    TEXT488 : BOOL ;	//TEXT N.488
    TEXT505 : BOOL ;	//TEXT N.505
    TEXT506 : BOOL ;	//TEXT N.506
    TEXT507 : BOOL ;	//TEXT N.507
    TEXT508 : BOOL ;	//TEXT N.508
    TEXT509 : BOOL ;	//TEXT N.509
    TEXT510 : BOOL ;	//TEXT N.510
    TEXT511 : BOOL ;	//TEXT N.511
    TEXT512 : BOOL ;	//TEXT N.512
    TEXT497 : BOOL ;	//TEXT N.497
    TEXT498 : BOOL ;	//TEXT N.498
    TEXT499 : BOOL ;	//TEXT N.499
    TEXT500 : BOOL ;	//TEXT N.500
    TEXT501 : BOOL ;	//TEXT N.501
    TEXT502 : BOOL ;	//TEXT N.502
    TEXT503 : BOOL ;	//TEXT N.503
    TEXT504 : BOOL ;	//TEXT N.504
    TEXT521 : BOOL ;	//TEXT N.521
    TEXT522 : BOOL ;	//TEXT N.522
    TEXT523 : BOOL ;	//TEXT N.523
    TEXT524 : BOOL ;	//TEXT N.524
    TEXT525 : BOOL ;	//TEXT N.525
    TEXT526 : BOOL ;	//TEXT N.526
    TEXT527 : BOOL ;	//TEXT N.527
    TEXT528 : BOOL ;	//TEXT N.528
    TEXT513 : BOOL ;	//TEXT N.513
    TEXT514 : BOOL ;	//TEXT N.514
    TEXT515 : BOOL ;	//TEXT N.515
    TEXT516 : BOOL ;	//TEXT N.516
    TEXT517 : BOOL ;	//TEXT N.517
    TEXT518 : BOOL ;	//TEXT N.518
    TEXT519 : BOOL ;	//TEXT N.519
    TEXT520 : BOOL ;	//TEXT N.520
    TEXT537 : BOOL ;	//TEXT N.537
    TEXT538 : BOOL ;	//TEXT N.538
    TEXT539 : BOOL ;	//TEXT N.539
    TEXT540 : BOOL ;	//TEXT N.540
    TEXT541 : BOOL ;	//TEXT N.541
    TEXT542 : BOOL ;	//TEXT N.542
    TEXT543 : BOOL ;	//TEXT N.543
    TEXT544 : BOOL ;	//TEXT N.544
    TEXT529 : BOOL ;	//TEXT N.529
    TEXT530 : BOOL ;	//TEXT N.530
    TEXT531 : BOOL ;	//TEXT N.531
    TEXT532 : BOOL ;	//TEXT N.532
    TEXT533 : BOOL ;	//TEXT N.533
    TEXT534 : BOOL ;	//TEXT N.534
    TEXT535 : BOOL ;	//TEXT N.535
    TEXT536 : BOOL ;	//TEXT N.536
    TEXT553 : BOOL ;	//TEXT N.553
    TEXT554 : BOOL ;	//TEXT N.554
    TEXT555 : BOOL ;	//TEXT N.555
    TEXT556 : BOOL ;	//TEXT N.556
    TEXT557 : BOOL ;	//TEXT N.557
    TEXT558 : BOOL ;	//TEXT N.558
    TEXT559 : BOOL ;	//TEXT N.559
    TEXT560 : BOOL ;	//TEXT N.560
    TEXT545 : BOOL ;	//TEXT N.545
    TEXT546 : BOOL ;	//TEXT N.546
    TEXT547 : BOOL ;	//TEXT N.547
    TEXT548 : BOOL ;	//TEXT N.548
    TEXT549 : BOOL ;	//TEXT N.549
    TEXT550 : BOOL ;	//TEXT N.550
    TEXT551 : BOOL ;	//TEXT N.551
    TEXT552 : BOOL ;	//TEXT N.552
    TEXT569 : BOOL ;	//TEXT N.569
    TEXT570 : BOOL ;	//TEXT N.570
    TEXT571 : BOOL ;	//TEXT N.571
    TEXT572 : BOOL ;	//TEXT N.572
    TEXT573 : BOOL ;	//TEXT N.573
    TEXT574 : BOOL ;	//TEXT N.574
    TEXT575 : BOOL ;	//TEXT N.575
    TEXT576 : BOOL ;	//TEXT N.576
    TEXT561 : BOOL ;	//TEXT N.561
    TEXT562 : BOOL ;	//TEXT N.562
    TEXT563 : BOOL ;	//TEXT N.563
    TEXT564 : BOOL ;	//TEXT N.564
    TEXT565 : BOOL ;	//TEXT N.565
    TEXT566 : BOOL ;	//TEXT N.566
    TEXT567 : BOOL ;	//TEXT N.567
    TEXT568 : BOOL ;	//TEXT N.568
    TEXT585 : BOOL ;	//TEXT N.585
    TEXT586 : BOOL ;	//TEXT N.586
    TEXT587 : BOOL ;	//TEXT N.587
    TEXT588 : BOOL ;	//TEXT N.588
    TEXT589 : BOOL ;	//TEXT N.589
    TEXT590 : BOOL ;	//TEXT N.590
    TEXT591 : BOOL ;	//TEXT N.591
    TEXT592 : BOOL ;	//TEXT N.592
    TEXT577 : BOOL ;	//TEXT N.577
    TEXT578 : BOOL ;	//TEXT N.578
    TEXT579 : BOOL ;	//TEXT N.579
    TEXT580 : BOOL ;	//TEXT N.580
    TEXT581 : BOOL ;	//TEXT N.581
    TEXT582 : BOOL ;	//TEXT N.582
    TEXT583 : BOOL ;	//TEXT N.583
    TEXT584 : BOOL ;	//TEXT N.584
    TEXT601 : BOOL ;	//TEXT N.601
    TEXT602 : BOOL ;	//TEXT N.602
    TEXT603 : BOOL ;	//TEXT N.603
    TEXT604 : BOOL ;	//TEXT N.604
    TEXT605 : BOOL ;	//TEXT N.605
    TEXT606 : BOOL ;	//TEXT N.606
    TEXT607 : BOOL ;	//TEXT N.607
    TEXT608 : BOOL ;	//TEXT N.608
    TEXT593 : BOOL ;	//TEXT N.593
    TEXT594 : BOOL ;	//TEXT N.594
    TEXT595 : BOOL ;	//TEXT N.595
    TEXT596 : BOOL ;	//TEXT N.596
    TEXT597 : BOOL ;	//TEXT N.597
    TEXT598 : BOOL ;	//TEXT N.598
    TEXT599 : BOOL ;	//TEXT N.599
    TEXT600 : BOOL ;	//TEXT N.600
    TEXT617 : BOOL ;	//TEXT N.617
    TEXT618 : BOOL ;	//TEXT N.618
    TEXT619 : BOOL ;	//TEXT N.619
    TEXT620 : BOOL ;	//TEXT N.620
    TEXT621 : BOOL ;	//TEXT N.621
    TEXT622 : BOOL ;	//TEXT N.622
    TEXT623 : BOOL ;	//TEXT N.623
    TEXT624 : BOOL ;	//TEXT N.624
    TEXT609 : BOOL ;	//TEXT N.609
    TEXT610 : BOOL ;	//TEXT N.610
    TEXT611 : BOOL ;	//TEXT N.611
    TEXT612 : BOOL ;	//TEXT N.612
    TEXT613 : BOOL ;	//TEXT N.613
    TEXT614 : BOOL ;	//TEXT N.614
    TEXT615 : BOOL ;	//TEXT N.615
    TEXT616 : BOOL ;	//TEXT N.616
    TEXT633 : BOOL ;	//TEXT N.633
    TEXT634 : BOOL ;	//TEXT N.634
    TEXT635 : BOOL ;	//TEXT N.635
    TEXT636 : BOOL ;	//TEXT N.636
    TEXT637 : BOOL ;	//TEXT N.637
    TEXT638 : BOOL ;	//TEXT N.638
    TEXT639 : BOOL ;	//TEXT N.639
    TEXT640 : BOOL ;	//TEXT N.640
    TEXT625 : BOOL ;	//TEXT N.625
    TEXT626 : BOOL ;	//TEXT N.626
    TEXT627 : BOOL ;	//TEXT N.627
    TEXT628 : BOOL ;	//TEXT N.628
    TEXT629 : BOOL ;	//TEXT N.629
    TEXT630 : BOOL ;	//TEXT N.630
    TEXT631 : BOOL ;	//TEXT N.631
    TEXT632 : BOOL ;	//TEXT N.632
   END_STRUCT ;
   PaginaDaVisualizzare : INT ;	//Number of page to display
   PaginaPrecedenteSetup : INT ;	//Number of page displayed before "Setup" page
   NumeroComandoManuale : INT ;	//Number of manual command
   BoschProgramManuale : BYTE ;	//Number of program of screwdriver in manual mode
   ServiceAsseSelezionato : BYTE ;	//Axis selected for movement in service mode (0=X; 1=Y; 2=Z; 3=C; 4=P)
   ServiceTipoJog : BYTE ;	//Kind of jog movement in service mode (0=continue; 1=incremental)
   ServiceFieldsDisplayed : BYTE ;	//Identify the fields to be displayed in service page
   TypePointTeachIn : BYTE ;	//Kind of screw in teach-in mode
   PointWeldingTeachIn : BYTE ;	//Identification of the screw in tech-in mode
   TeachInFieldsDisplayed : STRUCT 	//Identify the fields to be displayed in teach-in page
    Punto1Saldatura : BOOL ;
    Punto2Saldatura : BOOL ;
    Punto3Saldatura : BOOL ;
    Punto4Saldatura : BOOL ;
    Punto5Saldatura : BOOL ;
    Punto6Saldatura : BOOL ;
    Punto7Saldatura : BOOL ;
    Punto8Saldatura : BOOL ;
    Punto9Saldatura : BOOL ;
    Punto10Saldatura : BOOL ;
    Punto11Saldatura : BOOL ;
    Punto12Saldatura : BOOL ;
    Punto13Saldatura : BOOL ;
    PuntoVisione : BOOL ;
    Riserva1 : BOOL ;
    Riserva2 : BOOL ;
   END_STRUCT ;
   Target_Inc : DINT ;	//Target for the incremental movement
  END_STRUCT ;	
BEGIN
END_DATA_BLOCK

DATA_BLOCK DB 11
VERSION : 0.1
BEGIN
// 38 bytes; values not shown
END_DATA_BLOCK

DATA_BLOCK DB 12
VERSION : 0.1
BEGIN
// 38 bytes; values not shown
END_DATA_BLOCK

DATA_BLOCK DB 13
VERSION : 0.1
BEGIN
// 16 bytes; values not shown
END_DATA_BLOCK

DATA_BLOCK "Timer"	// DB 20
VERSION : 0.1
  STRUCT
   TmrOutGas : S5TIME  := S5T#1M;
   TmrIgnition : S5TIME  := S5T#20S;
   TmrDelayWelding : S5TIME  := S5T#300MS;
   time1 : S5TIME ;
   time11 : S5TIME ;
   time12 : S5TIME ;
   time13 : S5TIME ;
   time14 : S5TIME ;
   time15 : S5TIME ;
   time16 : S5TIME ;
   time17 : S5TIME ;
   time18 : S5TIME ;
   time19 : S5TIME ;
   time110 : S5TIME ;
   time111 : S5TIME ;
   time112 : S5TIME ;
   time113 : S5TIME ;
   time114 : S5TIME ;
   time115 : S5TIME ;
   time116 : S5TIME ;
   Override : INT  := 20;
   riserva2 : INT ;
   STAT22 : INT ;
   Comp01_OK : BOOL ;
   Comp02_OK : BOOL ;
   Comp03_OK : BOOL ;
   Comp04_OK : BOOL ;
   Comp05_OK : BOOL ;
   Comp06_OK : BOOL ;
   Comp07_OK : BOOL ;
   Comp08_OK : BOOL ;
   Comp09_OK : BOOL ;
   Comp10_OK : BOOL ;
   Comp11_OK : BOOL ;
   Comp12_OK : BOOL ;
   Comp13_OK : BOOL ;
   Comp14_OK : BOOL ;
   Comp15_OK : BOOL ;
   Comp16_OK : BOOL ;
   OffsetX1 : DINT ;
   OffsetY1 : DINT ;
   okAletta1 : BOOL ;
   okAletta2 : BOOL ;
   okAletta3 : BOOL ;
   okAletta4 : BOOL ;
   okAletta5 : BOOL ;
   okAletta6 : BOOL ;
   okAletta7 : BOOL ;
   okAletta8 : BOOL ;
   okAletta9 : BOOL ;
   okAletta10 : BOOL ;
   okAletta11 : BOOL ;
   okAletta12 : BOOL ;
   okAletta13 : BOOL ;
   okAletta14 : BOOL ;
   okAletta15 : BOOL ;
   okAletta16 : BOOL ;
   okAletta17 : BOOL ;
   okAletta18 : BOOL ;
   okAletta19 : BOOL ;
   okAletta20 : BOOL ;
   CheckComponent : BOOL  := TRUE;	//Check component with tool 1 --> Disable ; 0 --> Enable
   CheckTelec : BOOL ;	//Check Component with Omron 1 --> Disable ; 0 --> Enable
   check1 : BOOL ;
   CheckTelecafter : BOOL ;	//Check Component with Omron 1 --> Disable ; 0 --> Enable
   okAletta1_PP : BOOL ;
   okAletta2_PP : BOOL ;
   okAletta3_PP : BOOL ;
   okAletta4_PP : BOOL ;
   okAletta5_PP : BOOL ;
   okAletta6_PP : BOOL ;
   okAletta7_PP : BOOL ;
   okAletta8_PP : BOOL ;
   okAletta9_PP : BOOL ;
   okAletta10_PP : BOOL ;
   okAletta11_PP : BOOL ;
   okAletta12_PP : BOOL ;
   okAletta13_PP : BOOL ;
   okAletta14_PP : BOOL ;
   okAletta15_PP : BOOL ;
   okAletta16_PP : BOOL ;
   okAletta17_PP : BOOL ;
   okAletta18_PP : BOOL ;
   okAletta19_PP : BOOL ;
   okAletta20_PP : BOOL ;
   NumberVane : INT ;
   OffsetX2 : DINT ;
   OffsetY2 : DINT ;
  END_STRUCT ;	
BEGIN
   TmrOutGas := S5T#1M;
   TmrIgnition := S5T#20S;
   TmrDelayWelding := S5T#300MS;
   Override := 90;
   OffsetX1 := L#1550;
   OffsetY1 := L#-300;
   okAletta1 := TRUE;
   okAletta2 := TRUE;
   okAletta3 := TRUE;
   okAletta4 := TRUE;
   okAletta5 := TRUE;
   okAletta6 := TRUE;
   okAletta7 := TRUE;
   okAletta8 := TRUE;
   okAletta9 := TRUE;
   okAletta10 := TRUE;
   okAletta11 := TRUE;
   okAletta12 := TRUE;
   okAletta13 := TRUE;
   okAletta14 := TRUE;
   okAletta15 := TRUE;
   okAletta16 := TRUE;
   okAletta17 := TRUE;
   okAletta18 := TRUE;
   okAletta19 := TRUE;
   okAletta20 := TRUE;
   CheckComponent := TRUE;
   okAletta1_PP := TRUE;
   okAletta2_PP := TRUE;
   okAletta3_PP := TRUE;
   okAletta4_PP := TRUE;
   okAletta5_PP := TRUE;
   okAletta6_PP := TRUE;
   okAletta7_PP := TRUE;
   okAletta8_PP := TRUE;
   okAletta9_PP := TRUE;
   okAletta10_PP := TRUE;
   okAletta11_PP := TRUE;
   okAletta12_PP := TRUE;
   okAletta13_PP := TRUE;
   okAletta14_PP := TRUE;
   okAletta15_PP := TRUE;
   okAletta16_PP := TRUE;
   okAletta17_PP := TRUE;
   okAletta18_PP := TRUE;
   okAletta19_PP := TRUE;
   okAletta20_PP := TRUE;
   NumberVane := 2;
   OffsetX2 := L#1640;
   OffsetY2 := L#-400;
END_DATA_BLOCK

DATA_BLOCK "DBWork"	// DB 21
AUTHOR : Coletti
VERSION : 0.1
  STRUCT
   Famiglia : BYTE  := B#16#2;	//Type of family of product(2=Step2; 3=Step3)
   Turbo : BYTE  := B#16#1;	//Type of product
   Portapezzo1 : INT  := 1;	//Code of work rest 1
   Portapezzo2 : INT  := 1;	//Code of work rest 2
   TempoSaldatura : ARRAY  [1 .. 20 ] OF
   STRUCT
    Tempo : S5TIME  := S5T#1S;
   END_STRUCT ;
   CoordSaldatura : ARRAY  [1 .. 20 ] OF //Coordinates of points
   STRUCT
    X1 : DINT ;	//X coordinate of point
    Y1 : DINT ;	//Y coordinate of point
    X2 : DINT ;
    Y2 : DINT ;
   END_STRUCT ;
   EnableTelecamera : BOOL  := TRUE;
   PP : ARRAY  [1 .. 2 ] OF
   STRUCT
    Vuoto : BOOL ;
    Caricato : BOOL ;
    Bloccato : BOOL ;
    Fuori : BOOL ;
    Dentro : BOOL ;
    InLavorazione : BOOL ;
    Lavorato : BOOL ;
    Buobo : BOOL ;
    Scarto : BOOL ;
    NumSaldaturaAtt : INT ;
   END_STRUCT ;
   NumeroAnomalie : DINT ;
   NumeroPezziProd : DINT ;
   NumeroSaldature : INT ;
   Riserva : DINT ;
   Riserva1 : DINT ;
   RotationTable : BOOL ;	//angle rotation 1-->PP1 on welding; 0-->PP2 on Welding
   STAT29 : ARRAY  [1 .. 10 ] OF STRUCT
    x : DINT ;
    y : DINT ;
   END_STRUCT ;
   STAT32 : BYTE ;
   STAT33 : BYTE ;
  END_STRUCT ;	
BEGIN
   Famiglia := B#16#2;
   Turbo := B#16#1;
   Portapezzo1 := 1;
   Portapezzo2 := 1;
   TempoSaldatura[1].Tempo := S5T#1S700MS;
   TempoSaldatura[2].Tempo := S5T#1S350MS;
   TempoSaldatura[3].Tempo := S5T#1S;
   TempoSaldatura[4].Tempo := S5T#1S;
   TempoSaldatura[5].Tempo := S5T#1S;
   TempoSaldatura[6].Tempo := S5T#1S;
   TempoSaldatura[7].Tempo := S5T#1S;
   TempoSaldatura[8].Tempo := S5T#1S;
   TempoSaldatura[9].Tempo := S5T#1S;
   TempoSaldatura[10].Tempo := S5T#1S;
   TempoSaldatura[11].Tempo := S5T#1S;
   TempoSaldatura[12].Tempo := S5T#1S;
   TempoSaldatura[13].Tempo := S5T#1S;
   TempoSaldatura[14].Tempo := S5T#1S;
   TempoSaldatura[15].Tempo := S5T#1S;
   TempoSaldatura[16].Tempo := S5T#1S;
   TempoSaldatura[17].Tempo := S5T#1S;
   TempoSaldatura[18].Tempo := S5T#1S;
   TempoSaldatura[19].Tempo := S5T#1S;
   TempoSaldatura[20].Tempo := S5T#1S;
   CoordSaldatura[1].X1 := L#97555;
   CoordSaldatura[1].Y1 := L#158899;
   CoordSaldatura[1].X2 := L#97100;
   CoordSaldatura[1].Y2 := L#158948;
   CoordSaldatura[2].X1 := L#104046;
   CoordSaldatura[2].Y1 := L#174177;
   CoordSaldatura[2].X2 := L#103703;
   CoordSaldatura[2].Y2 := L#174196;
   CoordSaldatura[3].X1 := L#101148;
   CoordSaldatura[3].Y1 := L#190695;
   CoordSaldatura[3].X2 := L#100998;
   CoordSaldatura[3].Y2 := L#190806;
   CoordSaldatura[4].X1 := L#90048;
   CoordSaldatura[4].Y1 := L#202973;
   CoordSaldatura[4].X2 := L#89503;
   CoordSaldatura[4].Y2 := L#203030;
   CoordSaldatura[5].X1 := L#73999;
   CoordSaldatura[5].Y1 := L#207330;
   CoordSaldatura[5].X2 := L#73550;
   CoordSaldatura[5].Y2 := L#207355;
   CoordSaldatura[6].X1 := L#57802;
   CoordSaldatura[6].Y1 := L#202250;
   CoordSaldatura[6].X2 := L#57500;
   CoordSaldatura[6].Y2 := L#202334;
   CoordSaldatura[7].X1 := L#47102;
   CoordSaldatura[7].Y1 := L#189303;
   CoordSaldatura[7].X2 := L#46999;
   CoordSaldatura[7].Y2 := L#189221;
   CoordSaldatura[8].X1 := L#45249;
   CoordSaldatura[8].Y1 := L#172704;
   CoordSaldatura[8].X2 := L#44902;
   CoordSaldatura[8].Y2 := L#172596;
   CoordSaldatura[9].X1 := L#52600;
   CoordSaldatura[9].Y1 := L#157727;
   CoordSaldatura[9].X2 := L#52200;
   CoordSaldatura[9].Y2 := L#157808;
   CoordSaldatura[10].X1 := L#66950;
   CoordSaldatura[10].Y1 := L#149026;
   CoordSaldatura[10].X2 := L#66498;
   CoordSaldatura[10].Y2 := L#149001;
   CoordSaldatura[11].X1 := L#83750;
   CoordSaldatura[11].Y1 := L#149464;
   CoordSaldatura[11].X2 := L#83396;
   CoordSaldatura[11].Y2 := L#149500;
   EnableTelecamera := TRUE;
   NumeroSaldature := 11;
   RotationTable := TRUE;
   STAT29[1].x := L#124144;
   STAT29[1].y := L#141031;
END_DATA_BLOCK

DATA_BLOCK "coordinate"	// DB 22
VERSION : 0.1
  STRUCT
   CoordinatePP1 : ARRAY  [1 .. 20 ] OF
   STRUCT
    X1 : DINT ;
    Y1 : DINT ;
    X2 : DINT ;
    Y2 : DINT ;
   END_STRUCT ;
   CoordinatePP2 : ARRAY  [1 .. 20 ] OF
   STRUCT
    X1 : DINT ;
    Y1 : DINT ;
    X2 : DINT ;
    Y2 : DINT ;
   END_STRUCT ;
   STAT10 : ARRAY  [1 .. 20 ] OF STRUCT
    STAT11 : DINT ;
    STAT12 : DINT ;
    STAT13 : DINT ;
    STAT14 : DINT ;
   END_STRUCT ;
   STAT15 : ARRAY  [1 .. 20 ] OF STRUCT
    STAT16 : DINT ;
    STAT17 : DINT ;
    STAT18 : DINT ;
    STAT19 : DINT ;
   END_STRUCT ;
   STAT20 : ARRAY  [1 .. 20 ] OF STRUCT
    STAT21 : DINT ;
    STAT22 : DINT ;
    STAT23 : DINT ;
    STAT24 : DINT ;
   END_STRUCT ;
   STAT25 : ARRAY  [1 .. 20 ] OF STRUCT
    STAT26 : DINT ;
    STAT27 : DINT ;
    STAT28 : DINT ;
    STAT29 : DINT ;
   END_STRUCT ;
   STAT30 : ARRAY  [1 .. 20 ] OF STRUCT
    STAT31 : DINT ;
    STAT32 : DINT ;
    STAT33 : DINT ;
    STAT34 : DINT ;
   END_STRUCT ;
   STAT35 : ARRAY  [1 .. 20 ] OF STRUCT
    STAT36 : DINT ;
    STAT37 : DINT ;
    STAT38 : DINT ;
    STAT39 : DINT ;
   END_STRUCT ;
   STAT40 : ARRAY  [1 .. 20 ] OF STRUCT
    STAT41 : DINT ;
    STAT42 : DINT ;
    STAT43 : DINT ;
    STAT44 : DINT ;
   END_STRUCT ;
   STAT45 : ARRAY  [1 .. 20 ] OF STRUCT
    STAT46 : DINT ;
    STAT47 : DINT ;
    STAT48 : DINT ;
    STAT49 : DINT ;
   END_STRUCT ;
   STAT50 : ARRAY  [1 .. 20 ] OF STRUCT
    STAT51 : DINT ;
    STAT52 : DINT ;
    STAT53 : DINT ;
    STAT54 : DINT ;
   END_STRUCT ;
   STAT55 : ARRAY  [1 .. 20 ] OF STRUCT
    STAT56 : DINT ;
    STAT57 : DINT ;
    STAT58 : DINT ;
    STAT59 : DINT ;
   END_STRUCT ;
   STAT60 : ARRAY  [1 .. 20 ] OF STRUCT
    STAT61 : DINT ;
    STAT62 : DINT ;
    STAT63 : DINT ;
    STAT64 : DINT ;
   END_STRUCT ;
   STAT65 : ARRAY  [1 .. 20 ] OF STRUCT
    STAT66 : DINT ;
    STAT67 : DINT ;
    STAT68 : DINT ;
    STAT69 : DINT ;
   END_STRUCT ;
   STAT70 : ARRAY  [1 .. 20 ] OF STRUCT
    STAT71 : DINT ;
    STAT72 : DINT ;
    STAT73 : DINT ;
    STAT74 : DINT ;
   END_STRUCT ;
   STAT75 : ARRAY  [1 .. 20 ] OF STRUCT
    STAT76 : DINT ;
    STAT77 : DINT ;
    STAT78 : DINT ;
    STAT79 : DINT ;
   END_STRUCT ;
   STAT80 : ARRAY  [1 .. 20 ] OF STRUCT
    STAT81 : DINT ;
    STAT82 : DINT ;
    STAT83 : DINT ;
    STAT84 : DINT ;
   END_STRUCT ;
   STAT85 : ARRAY  [1 .. 20 ] OF STRUCT
    STAT86 : DINT ;
    STAT87 : DINT ;
    STAT88 : DINT ;
    STAT89 : DINT ;
   END_STRUCT ;
   STAT90 : ARRAY  [1 .. 20 ] OF STRUCT
    STAT91 : DINT ;
    STAT92 : DINT ;
    STAT93 : DINT ;
    STAT94 : DINT ;
   END_STRUCT ;
   STAT95 : ARRAY  [1 .. 20 ] OF STRUCT
    STAT96 : DINT ;
    STAT97 : DINT ;
    STAT98 : DINT ;
    STAT99 : DINT ;
   END_STRUCT ;
   STAT100 : ARRAY  [1 .. 10 ] OF STRUCT
    STAT101 : DINT ;
    STAT102 : DINT ;
   END_STRUCT ;
   STAT103 : ARRAY  [1 .. 10 ] OF STRUCT
    STAT104 : DINT ;
    STAT105 : DINT ;
   END_STRUCT ;
   STAT106 : ARRAY  [1 .. 10 ] OF STRUCT
    STAT107 : DINT ;
    STAT108 : DINT ;
   END_STRUCT ;
   STAT109 : ARRAY  [1 .. 10 ] OF STRUCT
    STAT110 : DINT ;
    STAT111 : DINT ;
   END_STRUCT ;
   STAT112 : ARRAY  [1 .. 10 ] OF STRUCT
    STAT113 : DINT ;
    STAT114 : DINT ;
   END_STRUCT ;
   STAT115 : ARRAY  [1 .. 10 ] OF STRUCT
    STAT116 : DINT ;
    STAT117 : DINT ;
   END_STRUCT ;
   STAT118 : ARRAY  [1 .. 10 ] OF STRUCT
    STAT119 : DINT ;
    STAT120 : DINT ;
   END_STRUCT ;
   STAT121 : ARRAY  [1 .. 10 ] OF STRUCT
    STAT122 : DINT ;
    STAT123 : DINT ;
   END_STRUCT ;
   STAT124 : ARRAY  [1 .. 10 ] OF STRUCT
    STAT125 : DINT ;
    STAT126 : DINT ;
   END_STRUCT ;
   STAT127 : ARRAY  [1 .. 10 ] OF STRUCT
    STAT128 : DINT ;
    STAT129 : DINT ;
   END_STRUCT ;
   STAT130 : ARRAY  [1 .. 10 ] OF STRUCT
    STAT131 : DINT ;
    STAT132 : DINT ;
   END_STRUCT ;
   STAT133 : ARRAY  [1 .. 10 ] OF STRUCT
    STAT134 : DINT ;
    STAT135 : DINT ;
   END_STRUCT ;
   STAT136 : ARRAY  [1 .. 10 ] OF STRUCT
    STAT137 : DINT ;
    STAT138 : DINT ;
   END_STRUCT ;
   STAT139 : ARRAY  [1 .. 10 ] OF STRUCT
    STAT140 : DINT ;
    STAT141 : DINT ;
   END_STRUCT ;
   STAT142 : ARRAY  [1 .. 10 ] OF STRUCT
    STAT143 : DINT ;
    STAT144 : DINT ;
   END_STRUCT ;
   STAT145 : ARRAY  [1 .. 10 ] OF STRUCT
    STAT146 : DINT ;
    STAT147 : DINT ;
   END_STRUCT ;
   STAT148 : ARRAY  [1 .. 10 ] OF STRUCT
    STAT149 : DINT ;
    STAT150 : DINT ;
   END_STRUCT ;
   STAT151 : ARRAY  [1 .. 10 ] OF STRUCT
    STAT152 : DINT ;
    STAT153 : DINT ;
   END_STRUCT ;
   STAT154 : ARRAY  [1 .. 10 ] OF STRUCT
    STAT155 : DINT ;
    STAT156 : DINT ;
   END_STRUCT ;
   STAT157 : ARRAY  [1 .. 10 ] OF STRUCT
    STAT158 : DINT ;
    STAT159 : DINT ;
   END_STRUCT ;
   STAT160 : INT ;
   STAT161 : INT ;
   STAT162 : INT ;
   STAT163 : INT ;
   STAT164 : INT ;
   STAT165 : INT ;
   STAT166 : INT ;
   STAT167 : INT ;
   STAT168 : INT ;
   STAT169 : INT ;
   STAT170 : INT ;
   STAT171 : INT ;
   STAT172 : INT ;
   STAT173 : INT ;
   STAT174 : INT ;
   STAT175 : INT ;
   STAT176 : INT ;
   STAT177 : INT ;
   STAT178 : INT ;
   STAT179 : INT ;
   STAT180 : ARRAY  [1 .. 20 ] OF STRUCT
    STAT181 : S5TIME  := S5T#1S;
   END_STRUCT ;
   STAT182 : ARRAY  [1 .. 20 ] OF STRUCT
    STAT183 : S5TIME  := S5T#1S;
   END_STRUCT ;
   STAT184 : ARRAY  [1 .. 20 ] OF STRUCT
    STAT185 : S5TIME  := S5T#1S;
   END_STRUCT ;
   STAT186 : ARRAY  [1 .. 20 ] OF STRUCT
    STAT187 : S5TIME  := S5T#1S;
   END_STRUCT ;
   STAT188 : ARRAY  [1 .. 20 ] OF STRUCT
    STAT189 : S5TIME  := S5T#1S;
   END_STRUCT ;
   STAT190 : ARRAY  [1 .. 20 ] OF STRUCT
    STAT191 : S5TIME  := S5T#1S;
   END_STRUCT ;
   STAT192 : ARRAY  [1 .. 20 ] OF STRUCT
    STAT193 : S5TIME  := S5T#1S;
   END_STRUCT ;
   STAT194 : ARRAY  [1 .. 20 ] OF STRUCT
    STAT195 : S5TIME  := S5T#1S;
   END_STRUCT ;
   STAT196 : ARRAY  [1 .. 20 ] OF STRUCT
    STAT197 : S5TIME  := S5T#1S;
   END_STRUCT ;
   STAT198 : ARRAY  [1 .. 20 ] OF STRUCT
    STAT199 : S5TIME  := S5T#1S;
   END_STRUCT ;
   STAT200 : ARRAY  [1 .. 20 ] OF STRUCT
    STAT201 : S5TIME  := S5T#1S;
   END_STRUCT ;
   STAT202 : ARRAY  [1 .. 20 ] OF STRUCT
    STAT203 : S5TIME  := S5T#1S;
   END_STRUCT ;
   STAT204 : ARRAY  [1 .. 20 ] OF STRUCT
    STAT205 : S5TIME  := S5T#1S;
   END_STRUCT ;
   STAT206 : ARRAY  [1 .. 20 ] OF STRUCT
    STAT207 : S5TIME  := S5T#1S;
   END_STRUCT ;
   STAT208 : ARRAY  [1 .. 20 ] OF STRUCT
    STAT209 : S5TIME  := S5T#1S;
   END_STRUCT ;
   STAT210 : ARRAY  [1 .. 20 ] OF STRUCT
    STAT211 : S5TIME  := S5T#1S;
   END_STRUCT ;
   STAT212 : ARRAY  [1 .. 20 ] OF STRUCT
    STAT213 : S5TIME  := S5T#1S;
   END_STRUCT ;
   STAT214 : ARRAY  [1 .. 20 ] OF STRUCT
    STAT215 : S5TIME  := S5T#1S;
   END_STRUCT ;
   STAT216 : ARRAY  [1 .. 20 ] OF STRUCT
    STAT217 : S5TIME  := S5T#1S;
   END_STRUCT ;
   STAT218 : ARRAY  [1 .. 20 ] OF STRUCT
    STAT219 : S5TIME  := S5T#1S;
   END_STRUCT ;
   STAT220 : BYTE ;
   STAT221 : BYTE ;
   STAT222 : BYTE ;
   STAT223 : BYTE ;
   STAT224 : BYTE ;
   STAT225 : BYTE ;
   STAT226 : BYTE ;
   STAT227 : BYTE ;
   STAT228 : BYTE ;
   STAT229 : BYTE ;
   STAT230 : BYTE ;
   STAT231 : BYTE ;
   STAT232 : BYTE ;
   STAT233 : BYTE ;
   STAT234 : BYTE ;
   STAT235 : BYTE ;
   STAT236 : BYTE ;
   STAT237 : BYTE ;
   STAT238 : BYTE ;
   STAT239 : BYTE ;
  END_STRUCT ;	
BEGIN
   CoordinatePP1[1].X1 := L#-60530;
   CoordinatePP1[1].Y1 := L#-172340;
   CoordinatePP1[1].X2 := L#-60530;
   CoordinatePP1[1].Y2 := L#-172340;
   CoordinatePP1[2].X1 := L#-46530;
   CoordinatePP1[2].Y1 := L#-162870;
   CoordinatePP1[2].X2 := L#-46530;
   CoordinatePP1[2].Y2 := L#-162870;
   CoordinatePP1[3].X1 := L#-29630;
   CoordinatePP1[3].Y1 := L#-163440;
   CoordinatePP1[3].X2 := L#-29630;
   CoordinatePP1[3].Y2 := L#-163440;
   CoordinatePP1[4].X1 := L#-16300;
   CoordinatePP1[4].Y1 := L#-173820;
   CoordinatePP1[4].X2 := L#-16300;
   CoordinatePP1[4].Y2 := L#-173820;
   CoordinatePP1[5].X1 := L#-11620;
   CoordinatePP1[5].Y1 := L#-190070;
   CoordinatePP1[5].X2 := L#-11620;
   CoordinatePP1[5].Y2 := L#-190070;
   CoordinatePP1[6].X1 := L#-17370;
   CoordinatePP1[6].Y1 := L#-205960;
   CoordinatePP1[6].X2 := L#-17370;
   CoordinatePP1[6].Y2 := L#-205960;
   CoordinatePP1[7].X1 := L#-31370;
   CoordinatePP1[7].Y1 := L#-215430;
   CoordinatePP1[7].X2 := L#-31370;
   CoordinatePP1[7].Y2 := L#-215430;
   CoordinatePP1[8].X1 := L#-48270;
   CoordinatePP1[8].Y1 := L#-214860;
   CoordinatePP1[8].X2 := L#-48270;
   CoordinatePP1[8].Y2 := L#-214860;
   CoordinatePP1[9].X1 := L#-61600;
   CoordinatePP1[9].Y1 := L#-204480;
   CoordinatePP1[9].X2 := L#-61600;
   CoordinatePP1[9].Y2 := L#-204480;
   CoordinatePP1[10].X1 := L#-66280;
   CoordinatePP1[10].Y1 := L#-188230;
   CoordinatePP1[10].X2 := L#-66280;
   CoordinatePP1[10].Y2 := L#-188230;
   CoordinatePP2[1].X1 := L#64310;
   CoordinatePP2[1].Y1 := L#227751;
   CoordinatePP2[1].X2 := L#63919;
   CoordinatePP2[1].Y2 := L#227365;
   CoordinatePP2[2].X1 := L#79927;
   CoordinatePP2[2].Y1 := L#232668;
   CoordinatePP2[2].X2 := L#79988;
   CoordinatePP2[2].Y2 := L#232846;
   CoordinatePP2[3].X1 := L#96108;
   CoordinatePP2[3].Y1 := L#228455;
   CoordinatePP2[3].X2 := L#95916;
   CoordinatePP2[3].Y2 := L#228643;
   CoordinatePP2[4].X1 := L#107420;
   CoordinatePP2[4].Y1 := L#216186;
   CoordinatePP2[4].X2 := L#107460;
   CoordinatePP2[4].Y2 := L#216344;
   CoordinatePP2[5].X1 := L#110315;
   CoordinatePP2[5].Y1 := L#199830;
   CoordinatePP2[5].X2 := L#110295;
   CoordinatePP2[5].Y2 := L#200118;
   CoordinatePP2[6].X1 := L#103824;
   CoordinatePP2[6].Y1 := L#184542;
   CoordinatePP2[6].X2 := L#103669;
   CoordinatePP2[6].Y2 := L#184630;
   CoordinatePP2[7].X1 := L#89911;
   CoordinatePP2[7].Y1 := L#175041;
   CoordinatePP2[7].X2 := L#89880;
   CoordinatePP2[7].Y2 := L#174907;
   CoordinatePP2[8].X1 := L#73442;
   CoordinatePP2[8].Y1 := L#174654;
   CoordinatePP2[8].X2 := L#73469;
   CoordinatePP2[8].Y2 := L#174722;
   CoordinatePP2[9].X1 := L#58789;
   CoordinatePP2[9].Y1 := L#182903;
   CoordinatePP2[9].X2 := L#59115;
   CoordinatePP2[9].Y2 := L#183380;
   STAT10[1].STAT11 := L#64310;
   STAT10[1].STAT12 := L#227751;
   STAT10[1].STAT13 := L#63919;
   STAT10[1].STAT14 := L#227365;
   STAT10[2].STAT11 := L#79927;
   STAT10[2].STAT12 := L#232668;
   STAT10[2].STAT13 := L#79988;
   STAT10[2].STAT14 := L#232846;
   STAT10[3].STAT11 := L#96108;
   STAT10[3].STAT12 := L#228455;
   STAT10[3].STAT13 := L#95916;
   STAT10[3].STAT14 := L#228643;
   STAT10[4].STAT11 := L#107420;
   STAT10[4].STAT12 := L#216186;
   STAT10[4].STAT13 := L#107460;
   STAT10[4].STAT14 := L#216344;
   STAT10[5].STAT11 := L#110315;
   STAT10[5].STAT12 := L#199830;
   STAT10[5].STAT13 := L#110295;
   STAT10[5].STAT14 := L#200118;
   STAT10[6].STAT11 := L#103824;
   STAT10[6].STAT12 := L#184542;
   STAT10[6].STAT13 := L#103669;
   STAT10[6].STAT14 := L#184630;
   STAT10[7].STAT11 := L#89911;
   STAT10[7].STAT12 := L#175041;
   STAT10[7].STAT13 := L#89880;
   STAT10[7].STAT14 := L#174907;
   STAT10[8].STAT11 := L#73442;
   STAT10[8].STAT12 := L#174654;
   STAT10[8].STAT13 := L#73469;
   STAT10[8].STAT14 := L#174722;
   STAT10[9].STAT11 := L#58789;
   STAT10[9].STAT12 := L#182903;
   STAT10[9].STAT13 := L#59115;
   STAT10[9].STAT14 := L#183380;
   STAT15[1].STAT16 := L#64310;
   STAT15[1].STAT17 := L#227751;
   STAT15[1].STAT18 := L#63919;
   STAT15[1].STAT19 := L#227365;
   STAT15[2].STAT16 := L#79927;
   STAT15[2].STAT17 := L#232668;
   STAT15[2].STAT18 := L#79988;
   STAT15[2].STAT19 := L#232846;
   STAT15[3].STAT16 := L#96108;
   STAT15[3].STAT17 := L#228455;
   STAT15[3].STAT18 := L#95916;
   STAT15[3].STAT19 := L#228643;
   STAT15[4].STAT16 := L#107420;
   STAT15[4].STAT17 := L#216186;
   STAT15[4].STAT18 := L#107460;
   STAT15[4].STAT19 := L#216344;
   STAT15[5].STAT16 := L#110315;
   STAT15[5].STAT17 := L#199830;
   STAT15[5].STAT18 := L#110295;
   STAT15[5].STAT19 := L#200118;
   STAT15[6].STAT16 := L#103824;
   STAT15[6].STAT17 := L#184542;
   STAT15[6].STAT18 := L#103669;
   STAT15[6].STAT19 := L#184630;
   STAT15[7].STAT16 := L#89911;
   STAT15[7].STAT17 := L#175041;
   STAT15[7].STAT18 := L#89880;
   STAT15[7].STAT19 := L#174907;
   STAT15[8].STAT16 := L#73442;
   STAT15[8].STAT17 := L#174654;
   STAT15[8].STAT18 := L#73469;
   STAT15[8].STAT19 := L#174722;
   STAT15[9].STAT16 := L#58789;
   STAT15[9].STAT17 := L#182903;
   STAT15[9].STAT18 := L#59115;
   STAT15[9].STAT19 := L#183380;
   STAT20[1].STAT21 := L#54000;
   STAT20[1].STAT22 := L#193598;
   STAT20[1].STAT23 := L#54328;
   STAT20[1].STAT24 := L#203650;
   STAT20[2].STAT21 := L#48350;
   STAT20[2].STAT22 := L#176001;
   STAT20[2].STAT23 := L#60113;
   STAT20[2].STAT24 := L#187750;
   STAT20[3].STAT21 := L#74650;
   STAT20[3].STAT22 := L#178100;
   STAT20[3].STAT23 := L#74400;
   STAT20[3].STAT24 := L#178249;
   STAT20[4].STAT21 := L#91766;
   STAT20[4].STAT22 := L#178750;
   STAT20[4].STAT23 := L#91450;
   STAT20[4].STAT24 := L#178950;
   STAT20[5].STAT21 := L#105100;
   STAT20[5].STAT22 := L#189150;
   STAT20[5].STAT23 := L#104730;
   STAT20[5].STAT24 := L#189300;
   STAT20[6].STAT21 := L#109714;
   STAT20[6].STAT22 := L#205845;
   STAT20[6].STAT23 := L#109290;
   STAT20[6].STAT24 := L#205700;
   STAT20[7].STAT21 := L#103650;
   STAT20[7].STAT22 := L#221740;
   STAT20[7].STAT23 := L#103470;
   STAT20[7].STAT24 := L#221801;
   STAT20[8].STAT21 := L#89526;
   STAT20[8].STAT22 := L#231180;
   STAT20[8].STAT23 := L#89330;
   STAT20[8].STAT24 := L#231180;
   STAT20[9].STAT21 := L#72660;
   STAT20[9].STAT22 := L#230570;
   STAT20[9].STAT23 := L#72209;
   STAT20[9].STAT24 := L#230560;
   STAT20[10].STAT21 := L#58901;
   STAT20[10].STAT22 := L#220019;
   STAT20[10].STAT23 := L#58901;
   STAT20[10].STAT24 := L#220019;
   STAT25[1].STAT26 := L#74397;
   STAT25[1].STAT27 := L#205796;
   STAT25[1].STAT28 := L#74886;
   STAT25[1].STAT29 := L#205247;
   STAT25[2].STAT26 := L#91400;
   STAT25[2].STAT27 := L#200192;
   STAT25[2].STAT28 := L#91897;
   STAT25[2].STAT29 := L#199346;
   STAT25[3].STAT26 := L#101849;
   STAT25[3].STAT27 := L#185291;
   STAT25[3].STAT28 := L#102145;
   STAT25[3].STAT29 := L#184898;
   STAT25[4].STAT26 := L#101897;
   STAT25[4].STAT27 := L#167497;
   STAT25[4].STAT28 := L#102300;
   STAT25[4].STAT29 := L#167046;
   STAT25[5].STAT26 := L#91097;
   STAT25[5].STAT27 := L#153097;
   STAT25[5].STAT28 := L#91299;
   STAT25[5].STAT29 := L#152598;
   STAT25[6].STAT26 := L#73999;
   STAT25[6].STAT27 := L#147792;
   STAT25[6].STAT28 := L#74002;
   STAT25[6].STAT29 := L#147077;
   STAT25[7].STAT26 := L#56999;
   STAT25[7].STAT27 := L#153695;
   STAT25[7].STAT28 := L#56949;
   STAT25[7].STAT29 := L#152781;
   STAT25[8].STAT26 := L#46396;
   STAT25[8].STAT27 := L#168197;
   STAT25[8].STAT28 := L#46449;
   STAT25[8].STAT29 := L#167745;
   STAT25[9].STAT26 := L#46395;
   STAT25[9].STAT27 := L#186097;
   STAT25[9].STAT28 := L#46698;
   STAT25[9].STAT29 := L#185745;
   STAT25[10].STAT26 := L#57199;
   STAT25[10].STAT27 := L#200597;
   STAT25[10].STAT28 := L#57697;
   STAT25[10].STAT29 := L#200145;
   STAT25[11].STAT26 := L#53800;
   STAT25[11].STAT27 := L#214850;
   STAT25[11].STAT28 := L#53936;
   STAT25[11].STAT29 := L#214811;
   STAT30[1].STAT31 := L#64310;
   STAT30[1].STAT32 := L#227751;
   STAT30[1].STAT33 := L#63919;
   STAT30[1].STAT34 := L#227365;
   STAT30[2].STAT31 := L#79927;
   STAT30[2].STAT32 := L#232668;
   STAT30[2].STAT33 := L#79988;
   STAT30[2].STAT34 := L#232846;
   STAT30[3].STAT31 := L#96108;
   STAT30[3].STAT32 := L#228455;
   STAT30[3].STAT33 := L#95916;
   STAT30[3].STAT34 := L#228643;
   STAT30[4].STAT31 := L#107420;
   STAT30[4].STAT32 := L#216186;
   STAT30[4].STAT33 := L#107460;
   STAT30[4].STAT34 := L#216344;
   STAT30[5].STAT31 := L#110315;
   STAT30[5].STAT32 := L#199830;
   STAT30[5].STAT33 := L#110295;
   STAT30[5].STAT34 := L#200118;
   STAT30[6].STAT31 := L#103824;
   STAT30[6].STAT32 := L#184542;
   STAT30[6].STAT33 := L#103669;
   STAT30[6].STAT34 := L#184630;
   STAT30[7].STAT31 := L#89911;
   STAT30[7].STAT32 := L#175041;
   STAT30[7].STAT33 := L#89880;
   STAT30[7].STAT34 := L#174907;
   STAT30[8].STAT31 := L#73442;
   STAT30[8].STAT32 := L#174654;
   STAT30[8].STAT33 := L#73469;
   STAT30[8].STAT34 := L#174722;
   STAT30[9].STAT31 := L#58789;
   STAT30[9].STAT32 := L#182903;
   STAT30[9].STAT33 := L#59115;
   STAT30[9].STAT34 := L#183380;
   STAT30[10].STAT31 := L#51760;
   STAT30[10].STAT32 := L#198339;
   STAT30[10].STAT33 := L#51980;
   STAT30[10].STAT34 := L#198401;
   STAT35[1].STAT36 := L#64510;
   STAT35[1].STAT37 := L#227751;
   STAT35[1].STAT38 := L#63919;
   STAT35[1].STAT39 := L#227365;
   STAT35[2].STAT36 := L#80000;
   STAT35[2].STAT37 := L#232720;
   STAT35[2].STAT38 := L#79988;
   STAT35[2].STAT39 := L#232846;
   STAT35[3].STAT36 := L#96250;
   STAT35[3].STAT37 := L#228455;
   STAT35[3].STAT38 := L#95916;
   STAT35[3].STAT39 := L#228643;
   STAT35[4].STAT36 := L#107420;
   STAT35[4].STAT37 := L#216186;
   STAT35[4].STAT38 := L#107460;
   STAT35[4].STAT39 := L#216344;
   STAT35[5].STAT36 := L#110315;
   STAT35[5].STAT37 := L#199830;
   STAT35[5].STAT38 := L#110295;
   STAT35[5].STAT39 := L#200118;
   STAT35[6].STAT36 := L#103824;
   STAT35[6].STAT37 := L#184542;
   STAT35[6].STAT38 := L#103669;
   STAT35[6].STAT39 := L#184630;
   STAT35[7].STAT36 := L#89911;
   STAT35[7].STAT37 := L#175041;
   STAT35[7].STAT38 := L#89880;
   STAT35[7].STAT39 := L#174907;
   STAT35[8].STAT36 := L#73442;
   STAT35[8].STAT37 := L#174654;
   STAT35[8].STAT38 := L#73469;
   STAT35[8].STAT39 := L#174722;
   STAT35[9].STAT36 := L#58789;
   STAT35[9].STAT37 := L#182903;
   STAT35[9].STAT38 := L#59115;
   STAT35[9].STAT39 := L#183380;
   STAT35[10].STAT36 := L#51760;
   STAT35[10].STAT37 := L#198339;
   STAT35[10].STAT38 := L#51980;
   STAT35[10].STAT39 := L#198401;
   STAT40[1].STAT41 := L#49300;
   STAT40[1].STAT42 := L#189673;
   STAT40[1].STAT43 := L#49568;
   STAT40[1].STAT44 := L#189634;
   STAT40[2].STAT41 := L#47551;
   STAT40[2].STAT42 := L#173065;
   STAT40[2].STAT43 := L#47627;
   STAT40[2].STAT44 := L#173198;
   STAT40[3].STAT41 := L#55179;
   STAT40[3].STAT42 := L#158249;
   STAT40[3].STAT43 := L#55080;
   STAT40[3].STAT44 := L#158254;
   STAT40[4].STAT41 := L#69324;
   STAT40[4].STAT42 := L#149465;
   STAT40[4].STAT43 := L#69322;
   STAT40[4].STAT44 := L#149454;
   STAT40[5].STAT41 := L#86091;
   STAT40[5].STAT42 := L#150123;
   STAT40[5].STAT43 := L#85999;
   STAT40[5].STAT44 := L#150019;
   STAT40[6].STAT41 := L#99264;
   STAT40[6].STAT42 := L#159144;
   STAT40[6].STAT43 := L#99400;
   STAT40[6].STAT44 := L#159195;
   STAT40[7].STAT41 := L#106332;
   STAT40[7].STAT42 := L#174551;
   STAT40[7].STAT43 := L#106482;
   STAT40[7].STAT44 := L#174661;
   STAT40[8].STAT41 := L#103460;
   STAT40[8].STAT42 := L#191130;
   STAT40[8].STAT43 := L#103553;
   STAT40[8].STAT44 := L#191049;
   STAT40[9].STAT41 := L#92009;
   STAT40[9].STAT42 := L#203434;
   STAT40[9].STAT43 := L#92323;
   STAT40[9].STAT44 := L#203330;
   STAT40[10].STAT41 := L#76002;
   STAT40[10].STAT42 := L#207802;
   STAT40[10].STAT43 := L#76052;
   STAT40[10].STAT44 := L#207819;
   STAT40[11].STAT41 := L#60002;
   STAT40[11].STAT42 := L#202602;
   STAT40[11].STAT43 := L#60303;
   STAT40[11].STAT44 := L#202658;
   STAT45[1].STAT46 := L#97555;
   STAT45[1].STAT47 := L#158899;
   STAT45[1].STAT48 := L#97100;
   STAT45[1].STAT49 := L#158948;
   STAT45[2].STAT46 := L#104046;
   STAT45[2].STAT47 := L#174177;
   STAT45[2].STAT48 := L#103703;
   STAT45[2].STAT49 := L#174196;
   STAT45[3].STAT46 := L#101148;
   STAT45[3].STAT47 := L#190695;
   STAT45[3].STAT48 := L#100998;
   STAT45[3].STAT49 := L#190806;
   STAT45[4].STAT46 := L#90048;
   STAT45[4].STAT47 := L#202973;
   STAT45[4].STAT48 := L#89503;
   STAT45[4].STAT49 := L#203030;
   STAT45[5].STAT46 := L#73999;
   STAT45[5].STAT47 := L#207330;
   STAT45[5].STAT48 := L#73550;
   STAT45[5].STAT49 := L#207355;
   STAT45[6].STAT46 := L#57802;
   STAT45[6].STAT47 := L#202250;
   STAT45[6].STAT48 := L#57500;
   STAT45[6].STAT49 := L#202334;
   STAT45[7].STAT46 := L#47102;
   STAT45[7].STAT47 := L#189303;
   STAT45[7].STAT48 := L#46999;
   STAT45[7].STAT49 := L#189221;
   STAT45[8].STAT46 := L#45249;
   STAT45[8].STAT47 := L#172704;
   STAT45[8].STAT48 := L#44902;
   STAT45[8].STAT49 := L#172596;
   STAT45[9].STAT46 := L#52600;
   STAT45[9].STAT47 := L#157727;
   STAT45[9].STAT48 := L#52200;
   STAT45[9].STAT49 := L#157808;
   STAT45[10].STAT46 := L#66950;
   STAT45[10].STAT47 := L#149026;
   STAT45[10].STAT48 := L#66498;
   STAT45[10].STAT49 := L#149001;
   STAT45[11].STAT46 := L#83750;
   STAT45[11].STAT47 := L#149464;
   STAT45[11].STAT48 := L#83396;
   STAT45[11].STAT49 := L#149500;
   STAT50[1].STAT51 := L#49591;
   STAT50[1].STAT52 := L#188786;
   STAT50[1].STAT53 := L#49492;
   STAT50[1].STAT54 := L#188701;
   STAT50[2].STAT51 := L#47690;
   STAT50[2].STAT52 := L#172414;
   STAT50[2].STAT53 := L#48025;
   STAT50[2].STAT54 := L#172138;
   STAT50[3].STAT51 := L#54723;
   STAT50[3].STAT52 := L#157462;
   STAT50[3].STAT53 := L#54578;
   STAT50[3].STAT54 := L#157545;
   STAT50[4].STAT51 := L#69395;
   STAT50[4].STAT52 := L#149104;
   STAT50[4].STAT53 := L#69105;
   STAT50[4].STAT54 := L#148974;
   STAT50[5].STAT51 := L#86010;
   STAT50[5].STAT52 := L#149692;
   STAT50[5].STAT53 := L#85816;
   STAT50[5].STAT54 := L#149590;
   STAT50[6].STAT51 := L#99522;
   STAT50[6].STAT52 := L#158915;
   STAT50[6].STAT53 := L#99438;
   STAT50[6].STAT54 := L#158302;
   STAT50[7].STAT51 := L#106030;
   STAT50[7].STAT52 := L#174316;
   STAT50[7].STAT53 := L#105672;
   STAT50[7].STAT54 := L#173776;
   STAT50[8].STAT51 := L#102900;
   STAT50[8].STAT52 := L#190978;
   STAT50[8].STAT53 := L#103227;
   STAT50[8].STAT54 := L#190062;
   STAT50[9].STAT51 := L#91916;
   STAT50[9].STAT52 := L#202939;
   STAT50[9].STAT53 := L#92233;
   STAT50[9].STAT54 := L#202347;
   STAT50[10].STAT51 := L#75327;
   STAT50[10].STAT52 := L#206920;
   STAT50[10].STAT53 := L#75993;
   STAT50[10].STAT54 := L#206482;
   STAT50[11].STAT51 := L#59823;
   STAT50[11].STAT52 := L#201921;
   STAT50[11].STAT53 := L#59921;
   STAT50[11].STAT54 := L#201602;
   STAT55[1].STAT56 := L#64310;
   STAT55[1].STAT57 := L#227751;
   STAT55[1].STAT58 := L#63919;
   STAT55[1].STAT59 := L#227365;
   STAT55[2].STAT56 := L#79927;
   STAT55[2].STAT57 := L#232668;
   STAT55[2].STAT58 := L#79988;
   STAT55[2].STAT59 := L#232846;
   STAT55[3].STAT56 := L#96108;
   STAT55[3].STAT57 := L#228455;
   STAT55[3].STAT58 := L#95916;
   STAT55[3].STAT59 := L#228643;
   STAT55[4].STAT56 := L#107420;
   STAT55[4].STAT57 := L#216186;
   STAT55[4].STAT58 := L#107460;
   STAT55[4].STAT59 := L#216344;
   STAT55[5].STAT56 := L#110315;
   STAT55[5].STAT57 := L#199830;
   STAT55[5].STAT58 := L#110295;
   STAT55[5].STAT59 := L#200118;
   STAT55[6].STAT56 := L#103824;
   STAT55[6].STAT57 := L#184542;
   STAT55[6].STAT58 := L#103669;
   STAT55[6].STAT59 := L#184630;
   STAT55[7].STAT56 := L#89911;
   STAT55[7].STAT57 := L#175041;
   STAT55[7].STAT58 := L#89880;
   STAT55[7].STAT59 := L#174907;
   STAT55[8].STAT56 := L#73442;
   STAT55[8].STAT57 := L#174654;
   STAT55[8].STAT58 := L#73469;
   STAT55[8].STAT59 := L#174722;
   STAT55[9].STAT56 := L#58789;
   STAT55[9].STAT57 := L#182903;
   STAT55[9].STAT58 := L#59115;
   STAT55[9].STAT59 := L#183380;
   STAT55[10].STAT56 := L#51760;
   STAT55[10].STAT57 := L#198339;
   STAT55[10].STAT58 := L#51980;
   STAT55[10].STAT59 := L#198401;
   STAT55[11].STAT56 := L#53800;
   STAT55[11].STAT57 := L#214850;
   STAT55[11].STAT58 := L#53936;
   STAT55[11].STAT59 := L#214811;
   STAT60[1].STAT61 := L#64310;
   STAT60[1].STAT62 := L#227751;
   STAT60[1].STAT63 := L#63919;
   STAT60[1].STAT64 := L#227365;
   STAT60[2].STAT61 := L#79927;
   STAT60[2].STAT62 := L#232668;
   STAT60[2].STAT63 := L#79988;
   STAT60[2].STAT64 := L#232846;
   STAT60[3].STAT61 := L#96108;
   STAT60[3].STAT62 := L#228455;
   STAT60[3].STAT63 := L#95916;
   STAT60[3].STAT64 := L#228643;
   STAT60[4].STAT61 := L#107420;
   STAT60[4].STAT62 := L#216186;
   STAT60[4].STAT63 := L#107460;
   STAT60[4].STAT64 := L#216344;
   STAT60[5].STAT61 := L#110315;
   STAT60[5].STAT62 := L#199830;
   STAT60[5].STAT63 := L#110295;
   STAT60[5].STAT64 := L#200118;
   STAT60[6].STAT61 := L#103824;
   STAT60[6].STAT62 := L#184542;
   STAT60[6].STAT63 := L#103669;
   STAT60[6].STAT64 := L#184630;
   STAT60[7].STAT61 := L#89911;
   STAT60[7].STAT62 := L#175041;
   STAT60[7].STAT63 := L#89880;
   STAT60[7].STAT64 := L#174907;
   STAT60[8].STAT61 := L#73442;
   STAT60[8].STAT62 := L#174654;
   STAT60[8].STAT63 := L#73469;
   STAT60[8].STAT64 := L#174722;
   STAT60[9].STAT61 := L#58789;
   STAT60[9].STAT62 := L#182903;
   STAT60[9].STAT63 := L#59115;
   STAT60[9].STAT64 := L#183380;
   STAT60[10].STAT61 := L#51760;
   STAT60[10].STAT62 := L#198339;
   STAT60[10].STAT63 := L#51980;
   STAT60[10].STAT64 := L#198401;
   STAT60[11].STAT61 := L#53800;
   STAT60[11].STAT62 := L#214850;
   STAT60[11].STAT63 := L#53936;
   STAT60[11].STAT64 := L#214811;
   STAT60[12].STAT61 := L#53800;
   STAT60[12].STAT62 := L#214850;
   STAT60[12].STAT63 := L#53936;
   STAT60[12].STAT64 := L#214811;
   STAT65[1].STAT66 := L#64310;
   STAT65[1].STAT67 := L#227751;
   STAT65[1].STAT68 := L#63919;
   STAT65[1].STAT69 := L#227365;
   STAT65[2].STAT66 := L#79927;
   STAT65[2].STAT67 := L#232668;
   STAT65[2].STAT68 := L#79988;
   STAT65[2].STAT69 := L#232846;
   STAT65[3].STAT66 := L#96108;
   STAT65[3].STAT67 := L#228455;
   STAT65[3].STAT68 := L#95916;
   STAT65[3].STAT69 := L#228643;
   STAT65[4].STAT66 := L#107420;
   STAT65[4].STAT67 := L#216186;
   STAT65[4].STAT68 := L#107460;
   STAT65[4].STAT69 := L#216344;
   STAT65[5].STAT66 := L#110315;
   STAT65[5].STAT67 := L#199830;
   STAT65[5].STAT68 := L#110295;
   STAT65[5].STAT69 := L#200118;
   STAT65[6].STAT66 := L#103824;
   STAT65[6].STAT67 := L#184542;
   STAT65[6].STAT68 := L#103669;
   STAT65[6].STAT69 := L#184630;
   STAT65[7].STAT66 := L#89911;
   STAT65[7].STAT67 := L#175041;
   STAT65[7].STAT68 := L#89880;
   STAT65[7].STAT69 := L#174907;
   STAT65[8].STAT66 := L#73442;
   STAT65[8].STAT67 := L#174654;
   STAT65[8].STAT68 := L#73469;
   STAT65[8].STAT69 := L#174722;
   STAT65[9].STAT66 := L#58789;
   STAT65[9].STAT67 := L#182903;
   STAT65[9].STAT68 := L#59115;
   STAT65[9].STAT69 := L#183380;
   STAT65[10].STAT66 := L#51760;
   STAT65[10].STAT67 := L#198339;
   STAT65[10].STAT68 := L#51980;
   STAT65[10].STAT69 := L#198401;
   STAT65[11].STAT66 := L#53800;
   STAT65[11].STAT67 := L#214850;
   STAT65[11].STAT68 := L#53936;
   STAT65[11].STAT69 := L#214811;
   STAT65[12].STAT66 := L#53800;
   STAT65[12].STAT67 := L#214850;
   STAT65[12].STAT68 := L#53936;
   STAT65[12].STAT69 := L#214811;
   STAT70[1].STAT71 := L#64310;
   STAT70[1].STAT72 := L#227751;
   STAT70[1].STAT73 := L#63919;
   STAT70[1].STAT74 := L#227365;
   STAT70[2].STAT71 := L#79927;
   STAT70[2].STAT72 := L#232668;
   STAT70[2].STAT73 := L#79988;
   STAT70[2].STAT74 := L#232846;
   STAT70[3].STAT71 := L#96108;
   STAT70[3].STAT72 := L#228455;
   STAT70[3].STAT73 := L#95916;
   STAT70[3].STAT74 := L#228643;
   STAT70[4].STAT71 := L#107420;
   STAT70[4].STAT72 := L#216186;
   STAT70[4].STAT73 := L#107460;
   STAT70[4].STAT74 := L#216344;
   STAT70[5].STAT71 := L#110315;
   STAT70[5].STAT72 := L#199830;
   STAT70[5].STAT73 := L#110295;
   STAT70[5].STAT74 := L#200118;
   STAT70[6].STAT71 := L#103824;
   STAT70[6].STAT72 := L#184542;
   STAT70[6].STAT73 := L#103669;
   STAT70[6].STAT74 := L#184630;
   STAT70[7].STAT71 := L#89911;
   STAT70[7].STAT72 := L#175041;
   STAT70[7].STAT73 := L#89880;
   STAT70[7].STAT74 := L#174907;
   STAT70[8].STAT71 := L#73442;
   STAT70[8].STAT72 := L#174654;
   STAT70[8].STAT73 := L#73469;
   STAT70[8].STAT74 := L#174722;
   STAT70[9].STAT71 := L#58789;
   STAT70[9].STAT72 := L#182903;
   STAT70[9].STAT73 := L#59115;
   STAT70[9].STAT74 := L#183380;
   STAT70[10].STAT71 := L#51760;
   STAT70[10].STAT72 := L#198339;
   STAT70[10].STAT73 := L#51980;
   STAT70[10].STAT74 := L#198401;
   STAT70[11].STAT71 := L#53800;
   STAT70[11].STAT72 := L#214850;
   STAT70[11].STAT73 := L#53936;
   STAT70[11].STAT74 := L#214811;
   STAT70[12].STAT71 := L#53800;
   STAT70[12].STAT72 := L#214850;
   STAT70[12].STAT73 := L#53936;
   STAT70[12].STAT74 := L#214811;
   STAT75[1].STAT76 := L#64310;
   STAT75[1].STAT77 := L#227751;
   STAT75[1].STAT78 := L#63919;
   STAT75[1].STAT79 := L#227365;
   STAT75[2].STAT76 := L#79927;
   STAT75[2].STAT77 := L#232668;
   STAT75[2].STAT78 := L#79988;
   STAT75[2].STAT79 := L#232846;
   STAT75[3].STAT76 := L#96108;
   STAT75[3].STAT77 := L#228455;
   STAT75[3].STAT78 := L#95916;
   STAT75[3].STAT79 := L#228643;
   STAT75[4].STAT76 := L#107420;
   STAT75[4].STAT77 := L#216186;
   STAT75[4].STAT78 := L#107460;
   STAT75[4].STAT79 := L#216344;
   STAT75[5].STAT76 := L#110315;
   STAT75[5].STAT77 := L#199830;
   STAT75[5].STAT78 := L#110295;
   STAT75[5].STAT79 := L#200118;
   STAT75[6].STAT76 := L#103824;
   STAT75[6].STAT77 := L#184542;
   STAT75[6].STAT78 := L#103669;
   STAT75[6].STAT79 := L#184630;
   STAT75[7].STAT76 := L#89911;
   STAT75[7].STAT77 := L#175041;
   STAT75[7].STAT78 := L#89880;
   STAT75[7].STAT79 := L#174907;
   STAT75[8].STAT76 := L#73442;
   STAT75[8].STAT77 := L#174654;
   STAT75[8].STAT78 := L#73469;
   STAT75[8].STAT79 := L#174722;
   STAT75[9].STAT76 := L#58789;
   STAT75[9].STAT77 := L#182903;
   STAT75[9].STAT78 := L#59115;
   STAT75[9].STAT79 := L#183380;
   STAT75[10].STAT76 := L#51760;
   STAT75[10].STAT77 := L#198339;
   STAT75[10].STAT78 := L#51980;
   STAT75[10].STAT79 := L#198401;
   STAT75[11].STAT76 := L#53800;
   STAT75[11].STAT77 := L#214850;
   STAT75[11].STAT78 := L#53936;
   STAT75[11].STAT79 := L#214811;
   STAT75[12].STAT76 := L#53800;
   STAT75[12].STAT77 := L#214850;
   STAT75[12].STAT78 := L#53936;
   STAT75[12].STAT79 := L#214811;
   STAT80[1].STAT81 := L#64310;
   STAT80[1].STAT82 := L#227751;
   STAT80[1].STAT83 := L#63919;
   STAT80[1].STAT84 := L#227365;
   STAT80[2].STAT81 := L#79927;
   STAT80[2].STAT82 := L#232668;
   STAT80[2].STAT83 := L#79988;
   STAT80[2].STAT84 := L#232846;
   STAT80[3].STAT81 := L#96108;
   STAT80[3].STAT82 := L#228455;
   STAT80[3].STAT83 := L#95916;
   STAT80[3].STAT84 := L#228643;
   STAT80[4].STAT81 := L#107420;
   STAT80[4].STAT82 := L#216186;
   STAT80[4].STAT83 := L#107460;
   STAT80[4].STAT84 := L#216344;
   STAT80[5].STAT81 := L#110315;
   STAT80[5].STAT82 := L#199830;
   STAT80[5].STAT83 := L#110295;
   STAT80[5].STAT84 := L#200118;
   STAT80[6].STAT81 := L#103824;
   STAT80[6].STAT82 := L#184542;
   STAT80[6].STAT83 := L#103669;
   STAT80[6].STAT84 := L#184630;
   STAT80[7].STAT81 := L#89911;
   STAT80[7].STAT82 := L#175041;
   STAT80[7].STAT83 := L#89880;
   STAT80[7].STAT84 := L#174907;
   STAT80[8].STAT81 := L#73442;
   STAT80[8].STAT82 := L#174654;
   STAT80[8].STAT83 := L#73469;
   STAT80[8].STAT84 := L#174722;
   STAT80[9].STAT81 := L#58789;
   STAT80[9].STAT82 := L#182903;
   STAT80[9].STAT83 := L#59115;
   STAT80[9].STAT84 := L#183380;
   STAT80[10].STAT81 := L#51760;
   STAT80[10].STAT82 := L#198339;
   STAT80[10].STAT83 := L#51980;
   STAT80[10].STAT84 := L#198401;
   STAT80[11].STAT81 := L#53800;
   STAT80[11].STAT82 := L#214850;
   STAT80[11].STAT83 := L#53936;
   STAT80[11].STAT84 := L#214811;
   STAT80[12].STAT81 := L#53800;
   STAT80[12].STAT82 := L#214850;
   STAT80[12].STAT83 := L#53936;
   STAT80[12].STAT84 := L#214811;
   STAT80[13].STAT81 := L#53800;
   STAT80[13].STAT82 := L#214850;
   STAT80[13].STAT83 := L#53936;
   STAT80[13].STAT84 := L#214811;
   STAT85[1].STAT86 := L#64310;
   STAT85[1].STAT87 := L#227751;
   STAT85[1].STAT88 := L#63919;
   STAT85[1].STAT89 := L#227365;
   STAT85[2].STAT86 := L#79927;
   STAT85[2].STAT87 := L#232668;
   STAT85[2].STAT88 := L#79988;
   STAT85[2].STAT89 := L#232846;
   STAT85[3].STAT86 := L#96108;
   STAT85[3].STAT87 := L#228455;
   STAT85[3].STAT88 := L#95916;
   STAT85[3].STAT89 := L#228643;
   STAT85[4].STAT86 := L#107420;
   STAT85[4].STAT87 := L#216186;
   STAT85[4].STAT88 := L#107460;
   STAT85[4].STAT89 := L#216344;
   STAT85[5].STAT86 := L#110315;
   STAT85[5].STAT87 := L#199830;
   STAT85[5].STAT88 := L#110295;
   STAT85[5].STAT89 := L#200118;
   STAT85[6].STAT86 := L#103824;
   STAT85[6].STAT87 := L#184542;
   STAT85[6].STAT88 := L#103669;
   STAT85[6].STAT89 := L#184630;
   STAT85[7].STAT86 := L#89911;
   STAT85[7].STAT87 := L#175041;
   STAT85[7].STAT88 := L#89880;
   STAT85[7].STAT89 := L#174907;
   STAT85[8].STAT86 := L#73442;
   STAT85[8].STAT87 := L#174654;
   STAT85[8].STAT88 := L#73469;
   STAT85[8].STAT89 := L#174722;
   STAT85[9].STAT86 := L#58789;
   STAT85[9].STAT87 := L#182903;
   STAT85[9].STAT88 := L#59115;
   STAT85[9].STAT89 := L#183380;
   STAT85[10].STAT86 := L#51760;
   STAT85[10].STAT87 := L#198339;
   STAT85[10].STAT88 := L#51980;
   STAT85[10].STAT89 := L#198401;
   STAT85[11].STAT86 := L#53800;
   STAT85[11].STAT87 := L#214850;
   STAT85[11].STAT88 := L#53936;
   STAT85[11].STAT89 := L#214811;
   STAT85[12].STAT86 := L#53800;
   STAT85[12].STAT87 := L#214850;
   STAT85[12].STAT88 := L#53936;
   STAT85[12].STAT89 := L#214811;
   STAT85[13].STAT86 := L#53800;
   STAT85[13].STAT87 := L#214850;
   STAT85[13].STAT88 := L#53936;
   STAT85[13].STAT89 := L#214811;
   STAT90[1].STAT91 := L#64310;
   STAT90[1].STAT92 := L#227751;
   STAT90[1].STAT93 := L#63919;
   STAT90[1].STAT94 := L#227365;
   STAT90[2].STAT91 := L#79927;
   STAT90[2].STAT92 := L#232668;
   STAT90[2].STAT93 := L#79988;
   STAT90[2].STAT94 := L#232846;
   STAT90[3].STAT91 := L#96108;
   STAT90[3].STAT92 := L#228455;
   STAT90[3].STAT93 := L#95916;
   STAT90[3].STAT94 := L#228643;
   STAT90[4].STAT91 := L#107420;
   STAT90[4].STAT92 := L#216186;
   STAT90[4].STAT93 := L#107460;
   STAT90[4].STAT94 := L#216344;
   STAT90[5].STAT91 := L#110315;
   STAT90[5].STAT92 := L#199830;
   STAT90[5].STAT93 := L#110295;
   STAT90[5].STAT94 := L#200118;
   STAT90[6].STAT91 := L#103824;
   STAT90[6].STAT92 := L#184542;
   STAT90[6].STAT93 := L#103669;
   STAT90[6].STAT94 := L#184630;
   STAT90[7].STAT91 := L#89911;
   STAT90[7].STAT92 := L#175041;
   STAT90[7].STAT93 := L#89880;
   STAT90[7].STAT94 := L#174907;
   STAT90[8].STAT91 := L#73442;
   STAT90[8].STAT92 := L#174654;
   STAT90[8].STAT93 := L#73469;
   STAT90[8].STAT94 := L#174722;
   STAT90[9].STAT91 := L#58789;
   STAT90[9].STAT92 := L#182903;
   STAT90[9].STAT93 := L#59115;
   STAT90[9].STAT94 := L#183380;
   STAT90[10].STAT91 := L#51760;
   STAT90[10].STAT92 := L#198339;
   STAT90[10].STAT93 := L#51980;
   STAT90[10].STAT94 := L#198401;
   STAT90[11].STAT91 := L#53800;
   STAT90[11].STAT92 := L#214850;
   STAT90[11].STAT93 := L#53936;
   STAT90[11].STAT94 := L#214811;
   STAT90[12].STAT91 := L#53800;
   STAT90[12].STAT92 := L#214850;
   STAT90[12].STAT93 := L#53936;
   STAT90[12].STAT94 := L#214811;
   STAT90[13].STAT91 := L#53800;
   STAT90[13].STAT92 := L#214850;
   STAT90[13].STAT93 := L#53936;
   STAT90[13].STAT94 := L#214811;
   STAT95[1].STAT96 := L#64310;
   STAT95[1].STAT97 := L#227751;
   STAT95[1].STAT98 := L#63919;
   STAT95[1].STAT99 := L#227365;
   STAT95[2].STAT96 := L#79927;
   STAT95[2].STAT97 := L#232668;
   STAT95[2].STAT98 := L#79988;
   STAT95[2].STAT99 := L#232846;
   STAT95[3].STAT96 := L#96108;
   STAT95[3].STAT97 := L#228455;
   STAT95[3].STAT98 := L#95916;
   STAT95[3].STAT99 := L#228643;
   STAT95[4].STAT96 := L#107420;
   STAT95[4].STAT97 := L#216186;
   STAT95[4].STAT98 := L#107460;
   STAT95[4].STAT99 := L#216344;
   STAT95[5].STAT96 := L#110315;
   STAT95[5].STAT97 := L#199830;
   STAT95[5].STAT98 := L#110295;
   STAT95[5].STAT99 := L#200118;
   STAT95[6].STAT96 := L#103824;
   STAT95[6].STAT97 := L#184542;
   STAT95[6].STAT98 := L#103669;
   STAT95[6].STAT99 := L#184630;
   STAT95[7].STAT96 := L#89911;
   STAT95[7].STAT97 := L#175041;
   STAT95[7].STAT98 := L#89880;
   STAT95[7].STAT99 := L#174907;
   STAT95[8].STAT96 := L#73442;
   STAT95[8].STAT97 := L#174654;
   STAT95[8].STAT98 := L#73469;
   STAT95[8].STAT99 := L#174722;
   STAT95[9].STAT96 := L#58789;
   STAT95[9].STAT97 := L#182903;
   STAT95[9].STAT98 := L#59115;
   STAT95[9].STAT99 := L#183380;
   STAT95[10].STAT96 := L#51760;
   STAT95[10].STAT97 := L#198339;
   STAT95[10].STAT98 := L#51980;
   STAT95[10].STAT99 := L#198401;
   STAT95[11].STAT96 := L#53800;
   STAT95[11].STAT97 := L#214850;
   STAT95[11].STAT98 := L#53936;
   STAT95[11].STAT99 := L#214811;
   STAT95[12].STAT96 := L#53800;
   STAT95[12].STAT97 := L#214850;
   STAT95[12].STAT98 := L#53936;
   STAT95[12].STAT99 := L#214811;
   STAT95[13].STAT96 := L#53800;
   STAT95[13].STAT97 := L#214850;
   STAT95[13].STAT98 := L#53936;
   STAT95[13].STAT99 := L#214811;
   STAT100[1].STAT101 := L#7915;
   STAT100[1].STAT102 := L#-68282;
   STAT103[1].STAT104 := L#124144;
   STAT103[1].STAT105 := L#141031;
   STAT106[1].STAT107 := L#124144;
   STAT106[1].STAT108 := L#141031;
   STAT109[1].STAT110 := L#124144;
   STAT109[1].STAT111 := L#141031;
   STAT112[1].STAT113 := L#124144;
   STAT112[1].STAT114 := L#141031;
   STAT115[1].STAT116 := L#124144;
   STAT115[1].STAT117 := L#141031;
   STAT118[1].STAT119 := L#124144;
   STAT118[1].STAT120 := L#141031;
   STAT121[1].STAT122 := L#124144;
   STAT121[1].STAT123 := L#141031;
   STAT124[1].STAT125 := L#101714;
   STAT124[1].STAT126 := L#142397;
   STAT127[1].STAT128 := L#124144;
   STAT127[1].STAT129 := L#141031;
   STAT130[1].STAT131 := L#124144;
   STAT130[1].STAT132 := L#141031;
   STAT133[1].STAT134 := L#124144;
   STAT133[1].STAT135 := L#141031;
   STAT136[1].STAT137 := L#124144;
   STAT136[1].STAT138 := L#141031;
   STAT139[1].STAT140 := L#124144;
   STAT139[1].STAT141 := L#141031;
   STAT142[1].STAT143 := L#124144;
   STAT142[1].STAT144 := L#141031;
   STAT145[1].STAT146 := L#124144;
   STAT145[1].STAT147 := L#141031;
   STAT148[1].STAT149 := L#124144;
   STAT148[1].STAT150 := L#141031;
   STAT151[1].STAT152 := L#124144;
   STAT151[1].STAT153 := L#141031;
   STAT154[1].STAT155 := L#124144;
   STAT154[1].STAT156 := L#141031;
   STAT157[1].STAT158 := L#124144;
   STAT157[1].STAT159 := L#141031;
   STAT160 := 10;
   STAT180[1].STAT181 := S5T#1S;
   STAT180[2].STAT181 := S5T#2S;
   STAT180[3].STAT181 := S5T#1S;
   STAT180[4].STAT181 := S5T#1S;
   STAT180[5].STAT181 := S5T#1S;
   STAT180[6].STAT181 := S5T#1S;
   STAT180[7].STAT181 := S5T#1S;
   STAT180[8].STAT181 := S5T#1S;
   STAT180[9].STAT181 := S5T#1S;
   STAT180[10].STAT181 := S5T#1S;
   STAT180[11].STAT181 := S5T#1S;
   STAT180[12].STAT181 := S5T#1S;
   STAT180[13].STAT181 := S5T#1S;
   STAT180[14].STAT181 := S5T#1S;
   STAT180[15].STAT181 := S5T#1S;
   STAT180[16].STAT181 := S5T#1S;
   STAT180[17].STAT181 := S5T#1S;
   STAT180[18].STAT181 := S5T#1S;
   STAT180[19].STAT181 := S5T#1S;
   STAT180[20].STAT181 := S5T#1S;
   STAT182[1].STAT183 := S5T#1S;
   STAT182[2].STAT183 := S5T#1S;
   STAT182[3].STAT183 := S5T#1S;
   STAT182[4].STAT183 := S5T#1S;
   STAT182[5].STAT183 := S5T#1S;
   STAT182[6].STAT183 := S5T#1S;
   STAT182[7].STAT183 := S5T#1S;
   STAT182[8].STAT183 := S5T#1S;
   STAT182[9].STAT183 := S5T#1S;
   STAT182[10].STAT183 := S5T#1S;
   STAT182[11].STAT183 := S5T#1S;
   STAT182[12].STAT183 := S5T#1S;
   STAT182[13].STAT183 := S5T#1S;
   STAT182[14].STAT183 := S5T#1S;
   STAT182[15].STAT183 := S5T#1S;
   STAT182[16].STAT183 := S5T#1S;
   STAT182[17].STAT183 := S5T#1S;
   STAT182[18].STAT183 := S5T#1S;
   STAT182[19].STAT183 := S5T#1S;
   STAT182[20].STAT183 := S5T#1S;
   STAT184[1].STAT185 := S5T#1S;
   STAT184[2].STAT185 := S5T#1S;
   STAT184[3].STAT185 := S5T#1S;
   STAT184[4].STAT185 := S5T#1S;
   STAT184[5].STAT185 := S5T#1S;
   STAT184[6].STAT185 := S5T#1S;
   STAT184[7].STAT185 := S5T#1S;
   STAT184[8].STAT185 := S5T#1S;
   STAT184[9].STAT185 := S5T#1S;
   STAT184[10].STAT185 := S5T#1S;
   STAT184[11].STAT185 := S5T#1S;
   STAT184[12].STAT185 := S5T#1S;
   STAT184[13].STAT185 := S5T#1S;
   STAT184[14].STAT185 := S5T#1S;
   STAT184[15].STAT185 := S5T#1S;
   STAT184[16].STAT185 := S5T#1S;
   STAT184[17].STAT185 := S5T#1S;
   STAT184[18].STAT185 := S5T#1S;
   STAT184[19].STAT185 := S5T#1S;
   STAT184[20].STAT185 := S5T#1S;
   STAT186[1].STAT187 := S5T#1S;
   STAT186[2].STAT187 := S5T#1S;
   STAT186[3].STAT187 := S5T#1S;
   STAT186[4].STAT187 := S5T#1S;
   STAT186[5].STAT187 := S5T#1S;
   STAT186[6].STAT187 := S5T#1S;
   STAT186[7].STAT187 := S5T#1S;
   STAT186[8].STAT187 := S5T#1S;
   STAT186[9].STAT187 := S5T#1S;
   STAT186[10].STAT187 := S5T#1S;
   STAT186[11].STAT187 := S5T#1S;
   STAT186[12].STAT187 := S5T#1S;
   STAT186[13].STAT187 := S5T#1S;
   STAT186[14].STAT187 := S5T#1S;
   STAT186[15].STAT187 := S5T#1S;
   STAT186[16].STAT187 := S5T#1S;
   STAT186[17].STAT187 := S5T#1S;
   STAT186[18].STAT187 := S5T#1S;
   STAT186[19].STAT187 := S5T#1S;
   STAT186[20].STAT187 := S5T#1S;
   STAT188[1].STAT189 := S5T#1S800MS;
   STAT188[2].STAT189 := S5T#1S350MS;
   STAT188[3].STAT189 := S5T#1S;
   STAT188[4].STAT189 := S5T#1S;
   STAT188[5].STAT189 := S5T#1S;
   STAT188[6].STAT189 := S5T#1S;
   STAT188[7].STAT189 := S5T#1S;
   STAT188[8].STAT189 := S5T#1S;
   STAT188[9].STAT189 := S5T#1S;
   STAT188[10].STAT189 := S5T#1S;
   STAT188[11].STAT189 := S5T#1S;
   STAT188[12].STAT189 := S5T#1S;
   STAT188[13].STAT189 := S5T#1S;
   STAT188[14].STAT189 := S5T#1S;
   STAT188[15].STAT189 := S5T#1S;
   STAT188[16].STAT189 := S5T#1S;
   STAT188[17].STAT189 := S5T#1S;
   STAT188[18].STAT189 := S5T#1S;
   STAT188[19].STAT189 := S5T#1S;
   STAT188[20].STAT189 := S5T#1S;
   STAT190[1].STAT191 := S5T#2S500MS;
   STAT190[2].STAT191 := S5T#2S;
   STAT190[3].STAT191 := S5T#1S;
   STAT190[4].STAT191 := S5T#1S;
   STAT190[5].STAT191 := S5T#1S;
   STAT190[6].STAT191 := S5T#1S;
   STAT190[7].STAT191 := S5T#1S;
   STAT190[8].STAT191 := S5T#1S;
   STAT190[9].STAT191 := S5T#1S;
   STAT190[10].STAT191 := S5T#1S;
   STAT190[11].STAT191 := S5T#1S;
   STAT190[12].STAT191 := S5T#1S;
   STAT190[13].STAT191 := S5T#1S;
   STAT190[14].STAT191 := S5T#1S;
   STAT190[15].STAT191 := S5T#1S;
   STAT190[16].STAT191 := S5T#1S;
   STAT190[17].STAT191 := S5T#1S;
   STAT190[18].STAT191 := S5T#1S;
   STAT190[19].STAT191 := S5T#1S;
   STAT190[20].STAT191 := S5T#1S;
   STAT192[1].STAT193 := S5T#1S;
   STAT192[2].STAT193 := S5T#1S;
   STAT192[3].STAT193 := S5T#1S;
   STAT192[4].STAT193 := S5T#1S;
   STAT192[5].STAT193 := S5T#1S;
   STAT192[6].STAT193 := S5T#1S;
   STAT192[7].STAT193 := S5T#1S;
   STAT192[8].STAT193 := S5T#1S;
   STAT192[9].STAT193 := S5T#1S;
   STAT192[10].STAT193 := S5T#1S;
   STAT192[11].STAT193 := S5T#1S;
   STAT192[12].STAT193 := S5T#1S;
   STAT192[13].STAT193 := S5T#1S;
   STAT192[14].STAT193 := S5T#1S;
   STAT192[15].STAT193 := S5T#1S;
   STAT192[16].STAT193 := S5T#1S;
   STAT192[17].STAT193 := S5T#1S;
   STAT192[18].STAT193 := S5T#1S;
   STAT192[19].STAT193 := S5T#1S;
   STAT192[20].STAT193 := S5T#1S;
   STAT194[1].STAT195 := S5T#1S;
   STAT194[2].STAT195 := S5T#1S;
   STAT194[3].STAT195 := S5T#1S;
   STAT194[4].STAT195 := S5T#1S;
   STAT194[5].STAT195 := S5T#1S;
   STAT194[6].STAT195 := S5T#1S;
   STAT194[7].STAT195 := S5T#1S;
   STAT194[8].STAT195 := S5T#1S;
   STAT194[9].STAT195 := S5T#1S;
   STAT194[10].STAT195 := S5T#1S;
   STAT194[11].STAT195 := S5T#1S;
   STAT194[12].STAT195 := S5T#1S;
   STAT194[13].STAT195 := S5T#1S;
   STAT194[14].STAT195 := S5T#1S;
   STAT194[15].STAT195 := S5T#1S;
   STAT194[16].STAT195 := S5T#1S;
   STAT194[17].STAT195 := S5T#1S;
   STAT194[18].STAT195 := S5T#1S;
   STAT194[19].STAT195 := S5T#1S;
   STAT194[20].STAT195 := S5T#1S;
   STAT196[1].STAT197 := S5T#1S700MS;
   STAT196[2].STAT197 := S5T#1S300MS;
   STAT196[3].STAT197 := S5T#1S;
   STAT196[4].STAT197 := S5T#1S;
   STAT196[5].STAT197 := S5T#1S;
   STAT196[6].STAT197 := S5T#1S;
   STAT196[7].STAT197 := S5T#1S;
   STAT196[8].STAT197 := S5T#1S;
   STAT196[9].STAT197 := S5T#1S;
   STAT196[10].STAT197 := S5T#1S;
   STAT196[11].STAT197 := S5T#1S;
   STAT196[12].STAT197 := S5T#1S;
   STAT196[13].STAT197 := S5T#1S;
   STAT196[14].STAT197 := S5T#1S;
   STAT196[15].STAT197 := S5T#1S;
   STAT196[16].STAT197 := S5T#1S;
   STAT196[17].STAT197 := S5T#1S;
   STAT196[18].STAT197 := S5T#1S;
   STAT196[19].STAT197 := S5T#1S;
   STAT196[20].STAT197 := S5T#1S;
   STAT198[1].STAT199 := S5T#1S700MS;
   STAT198[2].STAT199 := S5T#1S350MS;
   STAT198[3].STAT199 := S5T#1S;
   STAT198[4].STAT199 := S5T#1S;
   STAT198[5].STAT199 := S5T#1S;
   STAT198[6].STAT199 := S5T#1S;
   STAT198[7].STAT199 := S5T#1S;
   STAT198[8].STAT199 := S5T#1S;
   STAT198[9].STAT199 := S5T#1S;
   STAT198[10].STAT199 := S5T#1S;
   STAT198[11].STAT199 := S5T#1S;
   STAT198[12].STAT199 := S5T#1S;
   STAT198[13].STAT199 := S5T#1S;
   STAT198[14].STAT199 := S5T#1S;
   STAT198[15].STAT199 := S5T#1S;
   STAT198[16].STAT199 := S5T#1S;
   STAT198[17].STAT199 := S5T#1S;
   STAT198[18].STAT199 := S5T#1S;
   STAT198[19].STAT199 := S5T#1S;
   STAT198[20].STAT199 := S5T#1S;
   STAT200[1].STAT201 := S5T#1S;
   STAT200[2].STAT201 := S5T#1S;
   STAT200[3].STAT201 := S5T#1S;
   STAT200[4].STAT201 := S5T#1S;
   STAT200[5].STAT201 := S5T#1S;
   STAT200[6].STAT201 := S5T#1S;
   STAT200[7].STAT201 := S5T#1S;
   STAT200[8].STAT201 := S5T#1S;
   STAT200[9].STAT201 := S5T#1S;
   STAT200[10].STAT201 := S5T#1S;
   STAT200[11].STAT201 := S5T#1S;
   STAT200[12].STAT201 := S5T#1S;
   STAT200[13].STAT201 := S5T#1S;
   STAT200[14].STAT201 := S5T#1S;
   STAT200[15].STAT201 := S5T#1S;
   STAT200[16].STAT201 := S5T#1S;
   STAT200[17].STAT201 := S5T#1S;
   STAT200[18].STAT201 := S5T#1S;
   STAT200[19].STAT201 := S5T#1S;
   STAT200[20].STAT201 := S5T#1S;
   STAT202[1].STAT203 := S5T#1S;
   STAT202[2].STAT203 := S5T#1S;
   STAT202[3].STAT203 := S5T#1S;
   STAT202[4].STAT203 := S5T#1S;
   STAT202[5].STAT203 := S5T#1S;
   STAT202[6].STAT203 := S5T#1S;
   STAT202[7].STAT203 := S5T#1S;
   STAT202[8].STAT203 := S5T#1S;
   STAT202[9].STAT203 := S5T#1S;
   STAT202[10].STAT203 := S5T#1S;
   STAT202[11].STAT203 := S5T#1S;
   STAT202[12].STAT203 := S5T#1S;
   STAT202[13].STAT203 := S5T#1S;
   STAT202[14].STAT203 := S5T#1S;
   STAT202[15].STAT203 := S5T#1S;
   STAT202[16].STAT203 := S5T#1S;
   STAT202[17].STAT203 := S5T#1S;
   STAT202[18].STAT203 := S5T#1S;
   STAT202[19].STAT203 := S5T#1S;
   STAT202[20].STAT203 := S5T#1S;
   STAT204[1].STAT205 := S5T#1S;
   STAT204[2].STAT205 := S5T#1S;
   STAT204[3].STAT205 := S5T#1S;
   STAT204[4].STAT205 := S5T#1S;
   STAT204[5].STAT205 := S5T#1S;
   STAT204[6].STAT205 := S5T#1S;
   STAT204[7].STAT205 := S5T#1S;
   STAT204[8].STAT205 := S5T#1S;
   STAT204[9].STAT205 := S5T#1S;
   STAT204[10].STAT205 := S5T#1S;
   STAT204[11].STAT205 := S5T#1S;
   STAT204[12].STAT205 := S5T#1S;
   STAT204[13].STAT205 := S5T#1S;
   STAT204[14].STAT205 := S5T#1S;
   STAT204[15].STAT205 := S5T#1S;
   STAT204[16].STAT205 := S5T#1S;
   STAT204[17].STAT205 := S5T#1S;
   STAT204[18].STAT205 := S5T#1S;
   STAT204[19].STAT205 := S5T#1S;
   STAT204[20].STAT205 := S5T#1S;
   STAT206[1].STAT207 := S5T#1S;
   STAT206[2].STAT207 := S5T#1S;
   STAT206[3].STAT207 := S5T#1S;
   STAT206[4].STAT207 := S5T#1S;
   STAT206[5].STAT207 := S5T#1S;
   STAT206[6].STAT207 := S5T#1S;
   STAT206[7].STAT207 := S5T#1S;
   STAT206[8].STAT207 := S5T#1S;
   STAT206[9].STAT207 := S5T#1S;
   STAT206[10].STAT207 := S5T#1S;
   STAT206[11].STAT207 := S5T#1S;
   STAT206[12].STAT207 := S5T#1S;
   STAT206[13].STAT207 := S5T#1S;
   STAT206[14].STAT207 := S5T#1S;
   STAT206[15].STAT207 := S5T#1S;
   STAT206[16].STAT207 := S5T#1S;
   STAT206[17].STAT207 := S5T#1S;
   STAT206[18].STAT207 := S5T#1S;
   STAT206[19].STAT207 := S5T#1S;
   STAT206[20].STAT207 := S5T#1S;
   STAT208[1].STAT209 := S5T#1S;
   STAT208[2].STAT209 := S5T#1S;
   STAT208[3].STAT209 := S5T#1S;
   STAT208[4].STAT209 := S5T#1S;
   STAT208[5].STAT209 := S5T#1S;
   STAT208[6].STAT209 := S5T#1S;
   STAT208[7].STAT209 := S5T#1S;
   STAT208[8].STAT209 := S5T#1S;
   STAT208[9].STAT209 := S5T#1S;
   STAT208[10].STAT209 := S5T#1S;
   STAT208[11].STAT209 := S5T#1S;
   STAT208[12].STAT209 := S5T#1S;
   STAT208[13].STAT209 := S5T#1S;
   STAT208[14].STAT209 := S5T#1S;
   STAT208[15].STAT209 := S5T#1S;
   STAT208[16].STAT209 := S5T#1S;
   STAT208[17].STAT209 := S5T#1S;
   STAT208[18].STAT209 := S5T#1S;
   STAT208[19].STAT209 := S5T#1S;
   STAT208[20].STAT209 := S5T#1S;
   STAT210[1].STAT211 := S5T#1S;
   STAT210[2].STAT211 := S5T#1S;
   STAT210[3].STAT211 := S5T#1S;
   STAT210[4].STAT211 := S5T#1S;
   STAT210[5].STAT211 := S5T#1S;
   STAT210[6].STAT211 := S5T#1S;
   STAT210[7].STAT211 := S5T#1S;
   STAT210[8].STAT211 := S5T#1S;
   STAT210[9].STAT211 := S5T#1S;
   STAT210[10].STAT211 := S5T#1S;
   STAT210[11].STAT211 := S5T#1S;
   STAT210[12].STAT211 := S5T#1S;
   STAT210[13].STAT211 := S5T#1S;
   STAT210[14].STAT211 := S5T#1S;
   STAT210[15].STAT211 := S5T#1S;
   STAT210[16].STAT211 := S5T#1S;
   STAT210[17].STAT211 := S5T#1S;
   STAT210[18].STAT211 := S5T#1S;
   STAT210[19].STAT211 := S5T#1S;
   STAT210[20].STAT211 := S5T#1S;
   STAT212[1].STAT213 := S5T#1S;
   STAT212[2].STAT213 := S5T#1S;
   STAT212[3].STAT213 := S5T#1S;
   STAT212[4].STAT213 := S5T#1S;
   STAT212[5].STAT213 := S5T#1S;
   STAT212[6].STAT213 := S5T#1S;
   STAT212[7].STAT213 := S5T#1S;
   STAT212[8].STAT213 := S5T#1S;
   STAT212[9].STAT213 := S5T#1S;
   STAT212[10].STAT213 := S5T#1S;
   STAT212[11].STAT213 := S5T#1S;
   STAT212[12].STAT213 := S5T#1S;
   STAT212[13].STAT213 := S5T#1S;
   STAT212[14].STAT213 := S5T#1S;
   STAT212[15].STAT213 := S5T#1S;
   STAT212[16].STAT213 := S5T#1S;
   STAT212[17].STAT213 := S5T#1S;
   STAT212[18].STAT213 := S5T#1S;
   STAT212[19].STAT213 := S5T#1S;
   STAT212[20].STAT213 := S5T#1S;
   STAT214[1].STAT215 := S5T#1S;
   STAT214[2].STAT215 := S5T#1S;
   STAT214[3].STAT215 := S5T#1S;
   STAT214[4].STAT215 := S5T#1S;
   STAT214[5].STAT215 := S5T#1S;
   STAT214[6].STAT215 := S5T#1S;
   STAT214[7].STAT215 := S5T#1S;
   STAT214[8].STAT215 := S5T#1S;
   STAT214[9].STAT215 := S5T#1S;
   STAT214[10].STAT215 := S5T#1S;
   STAT214[11].STAT215 := S5T#1S;
   STAT214[12].STAT215 := S5T#1S;
   STAT214[13].STAT215 := S5T#1S;
   STAT214[14].STAT215 := S5T#1S;
   STAT214[15].STAT215 := S5T#1S;
   STAT214[16].STAT215 := S5T#1S;
   STAT214[17].STAT215 := S5T#1S;
   STAT214[18].STAT215 := S5T#1S;
   STAT214[19].STAT215 := S5T#1S;
   STAT214[20].STAT215 := S5T#1S;
   STAT216[1].STAT217 := S5T#1S;
   STAT216[2].STAT217 := S5T#1S;
   STAT216[3].STAT217 := S5T#1S;
   STAT216[4].STAT217 := S5T#1S;
   STAT216[5].STAT217 := S5T#1S;
   STAT216[6].STAT217 := S5T#1S;
   STAT216[7].STAT217 := S5T#1S;
   STAT216[8].STAT217 := S5T#1S;
   STAT216[9].STAT217 := S5T#1S;
   STAT216[10].STAT217 := S5T#1S;
   STAT216[11].STAT217 := S5T#1S;
   STAT216[12].STAT217 := S5T#1S;
   STAT216[13].STAT217 := S5T#1S;
   STAT216[14].STAT217 := S5T#1S;
   STAT216[15].STAT217 := S5T#1S;
   STAT216[16].STAT217 := S5T#1S;
   STAT216[17].STAT217 := S5T#1S;
   STAT216[18].STAT217 := S5T#1S;
   STAT216[19].STAT217 := S5T#1S;
   STAT216[20].STAT217 := S5T#1S;
   STAT218[1].STAT219 := S5T#1S;
   STAT218[2].STAT219 := S5T#1S;
   STAT218[3].STAT219 := S5T#1S;
   STAT218[4].STAT219 := S5T#1S;
   STAT218[5].STAT219 := S5T#1S;
   STAT218[6].STAT219 := S5T#1S;
   STAT218[7].STAT219 := S5T#1S;
   STAT218[8].STAT219 := S5T#1S;
   STAT218[9].STAT219 := S5T#1S;
   STAT218[10].STAT219 := S5T#1S;
   STAT218[11].STAT219 := S5T#1S;
   STAT218[12].STAT219 := S5T#1S;
   STAT218[13].STAT219 := S5T#1S;
   STAT218[14].STAT219 := S5T#1S;
   STAT218[15].STAT219 := S5T#1S;
   STAT218[16].STAT219 := S5T#1S;
   STAT218[17].STAT219 := S5T#1S;
   STAT218[18].STAT219 := S5T#1S;
   STAT218[19].STAT219 := S5T#1S;
   STAT218[20].STAT219 := S5T#1S;
END_DATA_BLOCK

DATA_BLOCK DB 23
VERSION : 0.1
BEGIN
// 2 bytes; values not shown
END_DATA_BLOCK

DATA_BLOCK "DB180"	// DB 180
VERSION : 0.0
"FB24 - Gestione Mov Assi"
BEGIN
END_DATA_BLOCK

DATA_BLOCK "DB181"	// DB 181
VERSION : 0.0
"FB24 - Gestione Mov Assi"
BEGIN
END_DATA_BLOCK

ORGANIZATION_BLOCK "MAIN PROGRAM"	// OB 1
VERSION : 0.1
VAR_TEMP
  TEMP0 : BYTE ;
  TEMP1 : BYTE ;
  TEMP2 : BYTE ;
  TEMP3 : BYTE ;
  TEMP4 : BYTE ;
  TEMP5 : BYTE ;
  TEMP6 : INT ;
  TEMP7 : INT ;
  TEMP8 : INT ;
  TEMP9 : DATE_AND_TIME ;
END_VAR
BEGIN
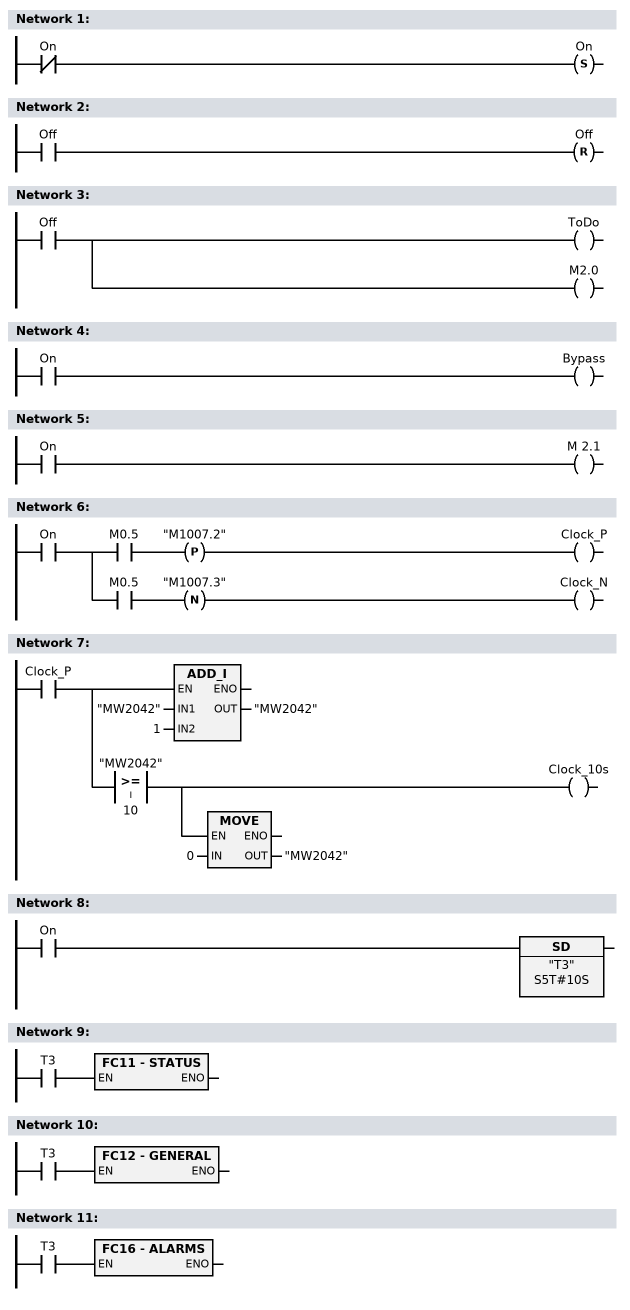
NETWORK
TITLE =
      AN    "On";
      S     "On";
NETWORK
TITLE =
      A     "Off";
      R     "Off";
NETWORK
TITLE =
      A     "Off";
      =     "ToDo";
      =     "M2.0";
NETWORK
TITLE =
      A     "On";
      =     "Bypass";
NETWORK
TITLE =
      A     "On";
      =     M 2.1;
NETWORK
TITLE =
      A     "On";
      =     L 20.0;
      A     L 20.0;
      A     "M0.5";
      FP    "M1007.2";
      =     "Clock_P";
      A     L 20.0;
      A     "M0.5";
      FN    "M1007.3";
      =     "Clock_N";
NETWORK
TITLE =
      A     "Clock_P";
      =     L 20.0;
      A     L 20.0;
      JNB   _001;
      L     "MW2042";
      L     1;
      +I;
      T     "MW2042";
_001: NOP   0;
      A     L 20.0;
      A(;
      L     "MW2042";
      L     10;
      >=I;
      );
      =     L 20.1;
      A     L 20.1;
      BLD   102;
      =     "Clock_10s";
      A     L 20.1;
      JNB   _002;
      L     0;
      T     "MW2042";
_002: NOP   0;
NETWORK
TITLE =
      A     "On";
      L     S5T#10S;
      SD    "T3";
NETWORK
TITLE =
      A     "T3";
      JNB   _003;
      CALL  "FC11 - STATUS";
_003: NOP   0;
NETWORK
TITLE =
      A     "T3";
      JNB   _004;
      CALL  "FC12 - GENERAL";
_004: NOP   0;
NETWORK
TITLE =
      A     "T3";
      JNB   _005;
      CALL  "FC16 - ALARMS";
_005: NOP   0;
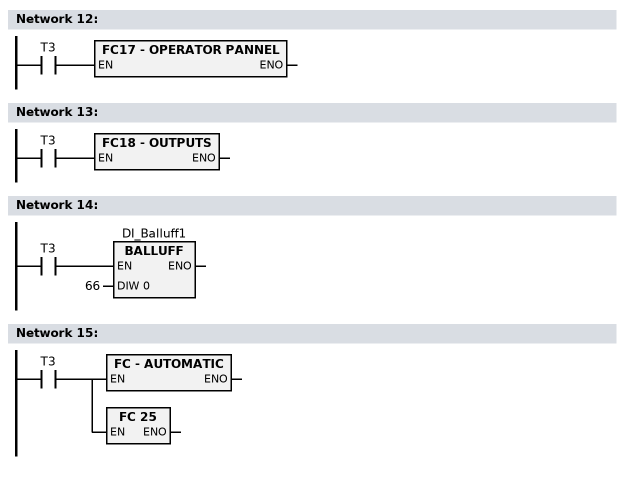
NETWORK
TITLE =
      A     "T3";
      JNB   _006;
      CALL  "FC17 - OPERATOR PANNEL";
_006: NOP   0;
NETWORK
TITLE =
      A     "T3";
      JNB   _007;
      CALL  "FC18 - OUTPUTS";
_007: NOP   0;
NETWORK
TITLE =
      A     "T3";
      JNB   _008;
      CALL  "BALLUFF" , "DI_Balluff1" (
           DIW 0                    := 66);
_008: NOP   0;
NETWORK
TITLE =
      A     "T3";
      =     L 20.0;
      A     L 20.0;
      JNB   _009;
      CALL  "FC - AUTOMATIC";
_009: NOP   0;
      A     L 20.0;
      JNB   _00a;
      CALL  FC 25;
_00a: NOP   0;
END_ORGANIZATION_BLOCK

ORGANIZATION_BLOCK "I/O_FLT1"	// OB 82
VERSION : 1.0
BEGIN
// (block stored without names or comments; labels and parameter names are numbered)
NETWORK
TITLE =
END_ORGANIZATION_BLOCK

ORGANIZATION_BLOCK "RACK_FLT"	// OB 86
VERSION : 0.1
BEGIN
// (block stored without names or comments; labels and parameter names are numbered)
NETWORK
TITLE =
END_ORGANIZATION_BLOCK

ORGANIZATION_BLOCK "COMPLETE RESTART"	// OB 100
VERSION : 0.1
BEGIN
// (block stored without names or comments; labels and parameter names are numbered)
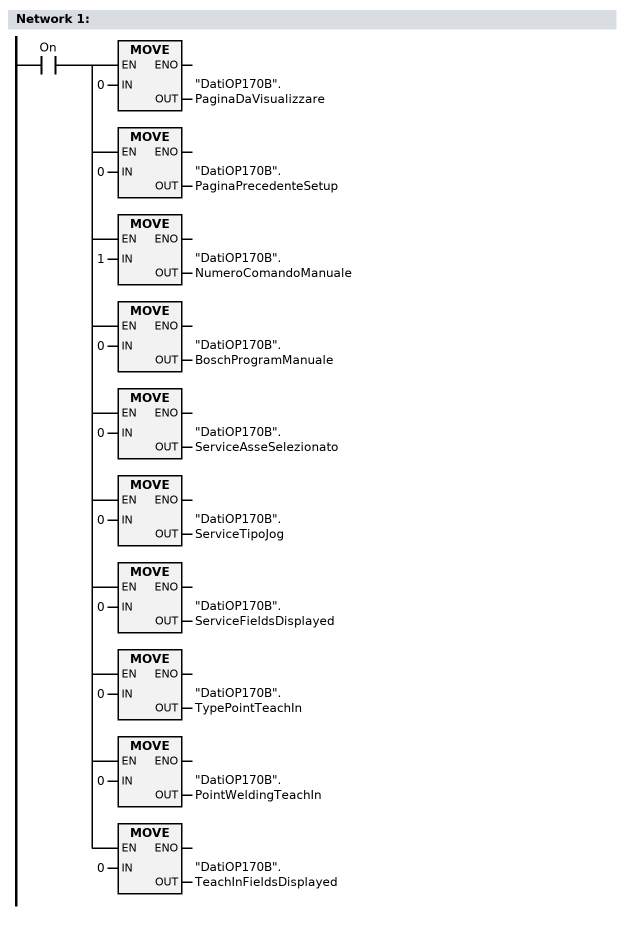
NETWORK
TITLE =
      A     "On";
      =     L 20.0;
      A     L 20.0;
      JNB   M001;
      L     0;
      T     "DatiOP170B".PaginaDaVisualizzare;
M001: NOP   0;
      A     L 20.0;
      JNB   M002;
      L     0;
      T     "DatiOP170B".PaginaPrecedenteSetup;
M002: NOP   0;
      A     L 20.0;
      JNB   M003;
      L     1;
      T     "DatiOP170B".NumeroComandoManuale;
M003: NOP   0;
      A     L 20.0;
      JNB   M004;
      L     0;
      T     "DatiOP170B".BoschProgramManuale;
M004: NOP   0;
      A     L 20.0;
      JNB   M005;
      L     0;
      T     "DatiOP170B".ServiceAsseSelezionato;
M005: NOP   0;
      A     L 20.0;
      JNB   M006;
      L     0;
      T     "DatiOP170B".ServiceTipoJog;
M006: NOP   0;
      A     L 20.0;
      JNB   M007;
      L     0;
      T     "DatiOP170B".ServiceFieldsDisplayed;
M007: NOP   0;
      A     L 20.0;
      JNB   M008;
      L     0;
      T     "DatiOP170B".TypePointTeachIn;
M008: NOP   0;
      A     L 20.0;
      JNB   M009;
      L     0;
      T     "DatiOP170B".PointWeldingTeachIn;
M009: NOP   0;
      A     L 20.0;
      JNB   M010;
      L     0;
      T     "DatiOP170B".TeachInFieldsDisplayed;
M010: NOP   0;
END_ORGANIZATION_BLOCK

ORGANIZATION_BLOCK "MOD_ERR"	// OB 122
VERSION : 0.1
BEGIN
// (block stored without names or comments; labels and parameter names are numbered)
NETWORK
TITLE =
END_ORGANIZATION_BLOCK

